  MoveL 7986 to (-27.4, 35.71, 116.27) mm, rotated rx 180 ry 0 rz 180 deg; joints [-139.207, -47.82, -97.335, 46.438, 64.37, -24.457]
  Call Extruder(71.60484)
  MoveL 7987 to (-27.15, 35.66, 116.27) mm, rotated rx 180 ry 0 rz -180 deg; joints [-139.239, -47.83, -97.308, 46.411, 64.345, -24.457]
  MoveL 7988 to (-27.15, 35.66, 116.27) mm, rotated rx 180 ry 0 rz -180 deg; joints [-139.239, -47.83, -97.308, 46.411, 64.345, -24.457]
  Call Extruder(71.75270)
  MoveL 7989 to (-26.87, 35.61, 116.27) mm, rotated rx -180 ry 0 rz -180 deg; joints [-139.275, -47.842, -97.278, 46.382, 64.317, -24.457]
  MoveL 7990 to (-26.87, 35.61, 116.27) mm, rotated rx -180 ry 0 rz -180 deg; joints [-139.275, -47.842, -97.278, 46.382, 64.317, -24.457]
  Call Extruder(71.91443)
  MoveL 7991 to (-26.57, 35.56, 116.27) mm, rotated rx 180 ry 0 rz 180 deg; joints [-139.313, -47.854, -97.243, 46.351, 64.286, -24.457]
  MoveL 7992 to (-26.57, 35.56, 116.27) mm, rotated rx 180 ry 0 rz 180 deg; joints [-139.313, -47.854, -97.243, 46.351, 64.286, -24.457]
  Call Extruder(72.07544)
  MoveL 7993 to (-26.26, 35.51, 116.27) mm, rotated rx 180 ry 0 rz 180 deg; joints [-139.351, -47.867, -97.209, 46.32, 64.255, -24.458]
  MoveL 7994 to (-26.26, 35.51, 116.27) mm, rotated rx 180 ry 0 rz 180 deg; joints [-139.351, -47.867, -97.209, 46.32, 64.255, -24.458]
  Call Extruder(72.23572)
  MoveL 7995 to (-25.96, 35.46, 116.27) mm, rotated rx 180 ry 0 rz -180 deg; joints [-139.39, -47.88, -97.174, 46.289, 64.225, -24.459]
  MoveL 7996 to (-25.96, 35.46, 116.27) mm, rotated rx 180 ry 0 rz -180 deg; joints [-139.39, -47.88, -97.174, 46.289, 64.225, -24.459]
  Call Extruder(72.39527)
  MoveL 7997 to (-25.65, 35.42, 116.27) mm, rotated rx 180 ry 0 rz 180 deg; joints [-139.428, -47.892, -97.14, 46.258, 64.194, -24.46]
  MoveL 7998 to (-25.65, 35.42, 116.27) mm, rotated rx 180 ry 0 rz 180 deg; joints [-139.428, -47.892, -97.14, 46.258, 64.194, -24.46]
  Call Extruder(72.55409)
  MoveL 7999 to (-25.34, 35.37, 116.27) mm, rotated rx 180 ry 0 rz -180 deg; joints [-139.466, -47.905, -97.105, 46.227, 64.163, -24.46]
  MoveL 8000 to (-25.34, 35.37, 116.27) mm, rotated rx 180 ry 0 rz -180 deg; joints [-139.466, -47.905, -97.105, 46.227, 64.163, -24.46]
  Call Extruder(72.73276)
  MoveL 8001 to (-25, 35.32, 116.27) mm, rotated rx 180 ry 0 rz -180 deg; joints [-139.508, -47.92, -97.065, 46.193, 64.128, -24.462]
  MoveL 8002 to (-25, 35.32, 116.27) mm, rotated rx 180 ry 0 rz -180 deg; joints [-139.508, -47.92, -97.065, 46.193, 64.128, -24.462]
  Call Extruder(72.93120)
  MoveL 8003 to (-24.61, 35.28, 116.27) mm, rotated rx 180 ry 0 rz 180 deg; joints [-139.554, -47.937, -97.019, 46.156, 64.089, -24.465]
  MoveL 8004 to (-24.61, 35.28, 116.27) mm, rotated rx 180 ry 0 rz 180 deg; joints [-139.554, -47.937, -97.019, 46.156, 64.089, -24.465]
  Call Extruder(73.12878)
  MoveL 8005 to (-24.22, 35.23, 116.27) mm, rotated rx 180 ry 0 rz 180 deg; joints [-139.6, -47.954, -96.973, 46.12, 64.05, -24.467]
  MoveL 8006 to (-24.22, 35.23, 116.27) mm, rotated rx 180 ry 0 rz 180 deg; joints [-139.6, -47.954, -96.973, 46.12, 64.05, -24.467]
  Call Extruder(73.32549)
  MoveL 8007 to (-23.84, 35.18, 116.27) mm, rotated rx -180 ry 0 rz 180 deg; joints [-139.647, -47.971, -96.928, 46.083, 64.01, -24.47]
  MoveL 8008 to (-23.84, 35.18, 116.27) mm, rotated rx -180 ry 0 rz 180 deg; joints [-139.647, -47.971, -96.928, 46.083, 64.01, -24.47]
  Call Extruder(73.52132)
  MoveL 8009 to (-23.45, 35.14, 116.27) mm, rotated rx 180 ry 0 rz 180 deg; joints [-139.693, -47.988, -96.882, 46.047, 63.971, -24.473]
  MoveL 8010 to (-23.45, 35.14, 116.27) mm, rotated rx 180 ry 0 rz 180 deg; joints [-139.693, -47.988, -96.882, 46.047, 63.971, -24.473]
  Call Extruder(73.81672)
  MoveL 8011 to (-22.86, 35.09, 116.27) mm, rotated rx 180 ry 0 rz -180 deg; joints [-139.76, -48.015, -96.809, 45.995, 63.912, -24.48]
  MoveL 8012 to (-22.86, 35.09, 116.27) mm, rotated rx 180 ry 0 rz -180 deg; joints [-139.76, -48.015, -96.809, 45.995, 63.912, -24.48]
  Call Extruder(74.11078)
  MoveL 8013 to (-22.27, 35.04, 116.27) mm, rotated rx -180 ry 0 rz -180 deg; joints [-139.826, -48.042, -96.736, 45.943, 63.852, -24.486]
  MoveL 8014 to (-22.27, 35.04, 116.27) mm, rotated rx -180 ry 0 rz -180 deg; joints [-139.826, -48.042, -96.736, 45.943, 63.852, -24.486]
  Call Extruder(74.40351)
  MoveL 8015 to (-21.68, 35, 116.27) mm, rotated rx 180 ry 0 rz 180 deg; joints [-139.893, -48.069, -96.664, 45.892, 63.793, -24.493]
  MoveL 8016 to (-21.68, 35, 116.27) mm, rotated rx 180 ry 0 rz 180 deg; joints [-139.893, -48.069, -96.664, 45.892, 63.793, -24.493]
  Call Extruder(74.97696)
  MoveL 8017 to (-20.52, 34.95, 116.27) mm, rotated rx 180 ry 0 rz -180 deg; joints [-140.019, -48.124, -96.515, 45.797, 63.675, -24.512]
  MoveL 8018 to (-20.52, 34.95, 116.27) mm, rotated rx 180 ry 0 rz -180 deg; joints [-140.019, -48.124, -96.515, 45.797, 63.675, -24.512]
  Call Extruder(75.69093)
  MoveL 8019 to (-19.06, 34.91, 116.27) mm, rotated rx 180 ry 0 rz 180 deg; joints [-140.173, -48.194, -96.326, 45.683, 63.529, -24.537]
  Call Extruder(192.53767)
  MoveL 8020 to (219.06, 34.91, 116.27) mm, rotated rx 180 ry 0 rz 180 deg; joints [-155.896, -66.609, -53.991, 41.312, 38.216, -34.626]
  Call Extruder(192.96623)
  MoveL 8021 to (219.94, 34.93, 116.27) mm, rotated rx 180 ry 0 rz -180 deg; joints [-155.931, -66.71, -53.779, 41.359, 38.112, -34.709]
  MoveL 8022 to (219.94, 34.93, 116.27) mm, rotated rx 180 ry 0 rz -180 deg; joints [-155.931, -66.71, -53.779, 41.359, 38.112, -34.709]
  Call Extruder(193.53967)
  MoveL 8023 to (221.1, 34.97, 116.27) mm, rotated rx 180 ry 0 rz 180 deg; joints [-155.975, -66.846, -53.494, 41.427, 37.975, -34.824]
  MoveL 8024 to (221.1, 34.97, 116.27) mm, rotated rx 180 ry 0 rz 180 deg; joints [-155.975, -66.846, -53.494, 41.427, 37.975, -34.824]
  Call Extruder(193.97399)
  MoveL 8025 to (221.97, 35.02, 116.27) mm, rotated rx 180 ry 0 rz 180 deg; joints [-156.007, -66.949, -53.276, 41.482, 37.871, -34.913]
  MoveL 8026 to (221.97, 35.02, 116.27) mm, rotated rx 180 ry 0 rz 180 deg; joints [-156.007, -66.949, -53.276, 41.482, 37.871, -34.913]
  Call Extruder(194.26805)
  MoveL 8027 to (222.56, 35.07, 116.27) mm, rotated rx -180 ry 0 rz -180 deg; joints [-156.027, -67.019, -53.128, 41.521, 37.802, -34.976]
  MoveL 8028 to (222.56, 35.07, 116.27) mm, rotated rx -180 ry 0 rz -180 deg; joints [-156.027, -67.019, -53.128, 41.521, 37.802, -34.976]
  Call Extruder(194.56344)
  MoveL 8029 to (223.15, 35.11, 116.27) mm, rotated rx 180 ry 0 rz 180 deg; joints [-156.047, -67.09, -52.98, 41.561, 37.732, -35.039]
  MoveL 8030 to (223.15, 35.11, 116.27) mm, rotated rx 180 ry 0 rz 180 deg; joints [-156.047, -67.09, -52.98, 41.561, 37.732, -35.039]
  Call Extruder(194.80967)
  MoveL 8031 to (223.64, 35.16, 116.27) mm, rotated rx 180 ry 0 rz 180 deg; joints [-156.062, -67.149, -52.855, 41.596, 37.674, -35.093]
  MoveL 8032 to (223.64, 35.16, 116.27) mm, rotated rx 180 ry 0 rz 180 deg; joints [-156.062, -67.149, -52.855, 41.596, 37.674, -35.093]
  Call Extruder(195.00638)
  MoveL 8033 to (224.03, 35.21, 116.27) mm, rotated rx 180 ry 0 rz 180 deg; joints [-156.074, -67.197, -52.756, 41.626, 37.628, -35.138]
  MoveL 8034 to (224.03, 35.21, 116.27) mm, rotated rx 180 ry 0 rz 180 deg; joints [-156.074, -67.197, -52.756, 41.626, 37.628, -35.138]
  Call Extruder(195.20395)
  MoveL 8035 to (224.42, 35.25, 116.27) mm, rotated rx -180 ry 0 rz 180 deg; joints [-156.086, -67.244, -52.656, 41.655, 37.583, -35.182]
  MoveL 8036 to (224.42, 35.25, 116.27) mm, rotated rx -180 ry 0 rz 180 deg; joints [-156.086, -67.244, -52.656, 41.655, 37.583, -35.182]
  Call Extruder(195.40240)
  MoveL 8037 to (224.8, 35.3, 116.27) mm, rotated rx 180 ry 0 rz 180 deg; joints [-156.097, -67.292, -52.556, 41.685, 37.537, -35.227]
  MoveL 8038 to (224.8, 35.3, 116.27) mm, rotated rx 180 ry 0 rz 180 deg; joints [-156.097, -67.292, -52.556, 41.685, 37.537, -35.227]
  Call Extruder(195.60171)
  MoveL 8039 to (225.19, 35.34, 116.27) mm, rotated rx 180 ry 0 rz 180 deg; joints [-156.109, -67.34, -52.456, 41.715, 37.491, -35.272]
  MoveL 8040 to (225.19, 35.34, 116.27) mm, rotated rx 180 ry 0 rz 180 deg; joints [-156.109, -67.34, -52.456, 41.715, 37.491, -35.272]
  Call Extruder(195.76053)
  MoveL 8041 to (225.5, 35.39, 116.27) mm, rotated rx 180 ry 0 rz 180 deg; joints [-156.117, -67.378, -52.375, 41.74, 37.455, -35.309]
  MoveL 8042 to (225.5, 35.39, 116.27) mm, rotated rx 180 ry 0 rz 180 deg; joints [-156.117, -67.378, -52.375, 41.74, 37.455, -35.309]
  Call Extruder(195.92007)
  MoveL 8043 to (225.8, 35.44, 116.27) mm, rotated rx 180 ry 0 rz 180 deg; joints [-156.125, -67.416, -52.295, 41.766, 37.419, -35.347]
  MoveL 8044 to (225.8, 35.44, 116.27) mm, rotated rx 180 ry 0 rz 180 deg; joints [-156.125, -67.416, -52.295, 41.766, 37.419, -35.347]
  Call Extruder(196.08035)
  MoveL 8045 to (226.11, 35.49, 116.27) mm, rotated rx 180 ry 0 rz 180 deg; joints [-156.133, -67.455, -52.214, 41.792, 37.383, -35.385]
  MoveL 8046 to (226.11, 35.49, 116.27) mm, rotated rx 180 ry 0 rz 180 deg; joints [-156.133, -67.455, -52.214, 41.792, 37.383, -35.385]
  Call Extruder(196.24135)
  MoveL 8047 to (226.41, 35.54, 116.27) mm, rotated rx -180 ry 0 rz -180 deg; joints [-156.141, -67.493, -52.133, 41.819, 37.347, -35.423]
  MoveL 8048 to (226.41, 35.54, 116.27) mm, rotated rx -180 ry 0 rz -180 deg; joints [-156.141, -67.493, -52.133, 41.819, 37.347, -35.423]
  Call Extruder(196.40308)
  MoveL 8049 to (226.72, 35.59, 116.27) mm, rotated rx -180 ry 0 rz -180 deg; joints [-156.149, -67.532, -52.053, 41.845, 37.311, -35.46]
  MoveL 8050 to (226.72, 35.59, 116.27) mm, rotated rx -180 ry 0 rz -180 deg; joints [-156.149, -67.532, -52.053, 41.845, 37.311, -35.46]
  Call Extruder(196.56554)
  MoveL 8051 to (227.03, 35.63, 116.27) mm, rotated rx -180 ry 0 rz 180 deg; joints [-156.157, -67.57, -51.972, 41.871, 37.275, -35.499]
  MoveL 8052 to (227.03, 35.63, 116.27) mm, rotated rx -180 ry 0 rz 180 deg; joints [-156.157, -67.57, -51.972, 41.871, 37.275, -35.499]
  Call Extruder(196.69947)
  MoveL 8053 to (227.28, 35.68, 116.27) mm, rotated rx 180 ry 0 rz 180 deg; joints [-156.162, -67.603, -51.905, 41.894, 37.245, -35.531]
  MoveL 8054 to (227.28, 35.68, 116.27) mm, rotated rx 180 ry 0 rz 180 deg; joints [-156.162, -67.603, -51.905, 41.894, 37.245, -35.531]
  Call Extruder(196.83401)
  MoveL 8055 to (227.52, 35.73, 116.27) mm, rotated rx -180 ry 0 rz -180 deg; joints [-156.168, -67.635, -51.837, 41.918, 37.216, -35.564]
  MoveL 8056 to (227.52, 35.73, 116.27) mm, rotated rx -180 ry 0 rz -180 deg; joints [-156.168, -67.635, -51.837, 41.918, 37.216, -35.564]
  Call Extruder(196.96915)
  MoveL 8057 to (227.77, 35.78, 116.27) mm, rotated rx 180 ry 0 rz -180 deg; joints [-156.173, -67.667, -51.77, 41.941, 37.186, -35.597]
  MoveL 8058 to (227.77, 35.78, 116.27) mm, rotated rx 180 ry 0 rz -180 deg; joints [-156.173, -67.667, -51.77, 41.941, 37.186, -35.597]
  Call Extruder(197.10491)
  MoveL 8059 to (228.02, 35.83, 116.27) mm, rotated rx 180 ry 0 rz 180 deg; joints [-156.179, -67.699, -51.703, 41.965, 37.157, -35.63]
  MoveL 8060 to (228.02, 35.83, 116.27) mm, rotated rx 180 ry 0 rz 180 deg; joints [-156.179, -67.699, -51.703, 41.965, 37.157, -35.63]
  Call Extruder(197.24128)
  MoveL 8061 to (228.27, 35.88, 116.27) mm, rotated rx 180 ry 0 rz 180 deg; joints [-156.185, -67.731, -51.636, 41.988, 37.128, -35.663]
  MoveL 8062 to (228.27, 35.88, 116.27) mm, rotated rx 180 ry 0 rz 180 deg; joints [-156.185, -67.731, -51.636, 41.988, 37.128, -35.663]
  Call Extruder(197.37826)
  MoveL 8063 to (228.52, 35.93, 116.27) mm, rotated rx -180 ry 0 rz 180 deg; joints [-156.19, -67.763, -51.568, 42.012, 37.098, -35.696]
  MoveL 8064 to (228.52, 35.93, 116.27) mm, rotated rx -180 ry 0 rz 180 deg; joints [-156.19, -67.763, -51.568, 42.012, 37.098, -35.696]
  Call Extruder(197.51585)
  MoveL 8065 to (228.77, 35.98, 116.27) mm, rotated rx 180 ry 0 rz 180 deg; joints [-156.196, -67.795, -51.501, 42.036, 37.069, -35.729]
  MoveL 8066 to (228.77, 35.98, 116.27) mm, rotated rx 180 ry 0 rz 180 deg; joints [-156.196, -67.795, -51.501, 42.036, 37.069, -35.729]
  Call Extruder(197.62957)
  MoveL 8067 to (228.97, 36.03, 116.27) mm, rotated rx 180 ry 0 rz 180 deg; joints [-156.2, -67.822, -51.445, 42.056, 37.045, -35.757]
  MoveL 8068 to (228.97, 36.03, 116.27) mm, rotated rx 180 ry 0 rz 180 deg; joints [-156.2, -67.822, -51.445, 42.056, 37.045, -35.757]
  Call Extruder(197.74374)
  MoveL 8069 to (229.18, 36.07, 116.27) mm, rotated rx -180 ry 0 rz 180 deg; joints [-156.204, -67.849, -51.389, 42.076, 37.021, -35.785]
  MoveL 8070 to (229.18, 36.07, 116.27) mm, rotated rx -180 ry 0 rz 180 deg; joints [-156.204, -67.849, -51.389, 42.076, 37.021, -35.785]
  Call Extruder(197.85836)
  MoveL 8071 to (229.38, 36.12, 116.27) mm, rotated rx -180 ry 0 rz 180 deg; joints [-156.208, -67.875, -51.333, 42.097, 36.997, -35.813]
  MoveL 8072 to (229.38, 36.12, 116.27) mm, rotated rx -180 ry 0 rz 180 deg; joints [-156.208, -67.875, -51.333, 42.097, 36.997, -35.813]
  Call Extruder(197.97344)
  MoveL 8073 to (229.59, 36.16, 116.27) mm, rotated rx 180 ry 0 rz 180 deg; joints [-156.212, -67.902, -51.277, 42.117, 36.973, -35.841]
  MoveL 8074 to (229.59, 36.16, 116.27) mm, rotated rx 180 ry 0 rz 180 deg; joints [-156.212, -67.902, -51.277, 42.117, 36.973, -35.841]
  Call Extruder(198.09430)
  MoveL 8075 to (229.8, 36.21, 116.27) mm, rotated rx -180 ry 0 rz 180 deg; joints [-156.216, -67.93, -51.218, 42.14, 36.948, -35.872]
  MoveL 8076 to (229.8, 36.21, 116.27) mm, rotated rx -180 ry 0 rz 180 deg; joints [-156.216, -67.93, -51.218, 42.14, 36.948, -35.872]
  Call Extruder(198.22115)
  MoveL 8077 to (230.02, 36.28, 116.27) mm, rotated rx -180 ry 0 rz -180 deg; joints [-156.219, -67.96, -51.156, 42.165, 36.922, -35.905]
  MoveL 8078 to (230.02, 36.28, 116.27) mm, rotated rx -180 ry 0 rz -180 deg; joints [-156.219, -67.96, -51.156, 42.165, 36.922, -35.905]
  Call Extruder(198.33995)
  MoveL 8079 to (230.22, 36.34, 116.27) mm, rotated rx -180 ry 0 rz -180 deg; joints [-156.222, -67.988, -51.098, 42.188, 36.898, -35.936]
  MoveL 8080 to (230.22, 36.34, 116.27) mm, rotated rx -180 ry 0 rz -180 deg; joints [-156.222, -67.988, -51.098, 42.188, 36.898, -35.936]
  Call Extruder(198.45066)
  MoveL 8081 to (230.41, 36.4, 116.27) mm, rotated rx -180 ry 0 rz -180 deg; joints [-156.224, -68.014, -51.044, 42.21, 36.876, -35.965]
  MoveL 8082 to (230.41, 36.4, 116.27) mm, rotated rx -180 ry 0 rz -180 deg; joints [-156.224, -68.014, -51.044, 42.21, 36.876, -35.965]
  Call Extruder(198.56179)
  MoveL 8083 to (230.6, 36.46, 116.27) mm, rotated rx 180 ry 0 rz -180 deg; joints [-156.226, -68.039, -50.99, 42.232, 36.854, -35.994]
  MoveL 8084 to (230.6, 36.46, 116.27) mm, rotated rx 180 ry 0 rz -180 deg; joints [-156.226, -68.039, -50.99, 42.232, 36.854, -35.994]
  Call Extruder(198.67341)
  MoveL 8085 to (230.79, 36.52, 116.27) mm, rotated rx 180 ry 0 rz 180 deg; joints [-156.228, -68.065, -50.936, 42.255, 36.831, -36.023]
  MoveL 8086 to (230.79, 36.52, 116.27) mm, rotated rx 180 ry 0 rz 180 deg; joints [-156.228, -68.065, -50.936, 42.255, 36.831, -36.023]
  Call Extruder(198.78553)
  MoveL 8087 to (230.98, 36.58, 116.27) mm, rotated rx 180 ry 0 rz 180 deg; joints [-156.23, -68.091, -50.882, 42.278, 36.809, -36.053]
  MoveL 8088 to (230.98, 36.58, 116.27) mm, rotated rx 180 ry 0 rz 180 deg; joints [-156.23, -68.091, -50.882, 42.278, 36.809, -36.053]
  Call Extruder(198.89810)
  MoveL 8089 to (231.17, 36.64, 116.27) mm, rotated rx -180 ry 0 rz 180 deg; joints [-156.232, -68.117, -50.828, 42.3, 36.787, -36.082]
  MoveL 8090 to (231.17, 36.64, 116.27) mm, rotated rx -180 ry 0 rz 180 deg; joints [-156.232, -68.117, -50.828, 42.3, 36.787, -36.082]
  Call Extruder(199.01111)
  MoveL 8091 to (231.35, 36.7, 116.27) mm, rotated rx -180 ry 0 rz 180 deg; joints [-156.234, -68.143, -50.774, 42.323, 36.765, -36.112]
  MoveL 8092 to (231.35, 36.7, 116.27) mm, rotated rx -180 ry 0 rz 180 deg; joints [-156.234, -68.143, -50.774, 42.323, 36.765, -36.112]
  Call Extruder(199.12456)
  MoveL 8093 to (231.54, 36.76, 116.27) mm, rotated rx 180 ry 0 rz -180 deg; joints [-156.236, -68.169, -50.719, 42.346, 36.743, -36.142]
  MoveL 8094 to (231.54, 36.76, 116.27) mm, rotated rx 180 ry 0 rz -180 deg; joints [-156.236, -68.169, -50.719, 42.346, 36.743, -36.142]
  Call Extruder(199.27220)
  MoveL 8095 to (231.78, 36.85, 116.27) mm, rotated rx -180 ry 0 rz 180 deg; joints [-156.237, -68.203, -50.649, 42.378, 36.715, -36.182]
  MoveL 8096 to (231.78, 36.85, 116.27) mm, rotated rx -180 ry 0 rz 180 deg; joints [-156.237, -68.203, -50.649, 42.378, 36.715, -36.182]
  Call Extruder(199.45454)
  MoveL 8097 to (232.07, 36.97, 116.27) mm, rotated rx -180 ry 0 rz 180 deg; joints [-156.238, -68.245, -50.562, 42.418, 36.681, -36.232]
  MoveL 8098 to (232.07, 36.97, 116.27) mm, rotated rx -180 ry 0 rz 180 deg; joints [-156.238, -68.245, -50.562, 42.418, 36.681, -36.232]
  Call Extruder(199.63764)
  MoveL 8099 to (232.37, 37.09, 116.27) mm, rotated rx -180 ry 0 rz 180 deg; joints [-156.239, -68.286, -50.474, 42.458, 36.647, -36.283]
  MoveL 8100 to (232.37, 37.09, 116.27) mm, rotated rx -180 ry 0 rz 180 deg; joints [-156.239, -68.286, -50.474, 42.458, 36.647, -36.283]
  Call Extruder(199.79534)
  MoveL 8101 to (232.62, 37.2, 116.27) mm, rotated rx 180 ry 0 rz 180 deg; joints [-156.239, -68.322, -50.399, 42.493, 36.618, -36.327]
  MoveL 8102 to (232.62, 37.2, 116.27) mm, rotated rx 180 ry 0 rz 180 deg; joints [-156.239, -68.322, -50.399, 42.493, 36.618, -36.327]
  Call Extruder(199.95364)
  MoveL 8103 to (232.86, 37.31, 116.27) mm, rotated rx 180 ry 0 rz 180 deg; joints [-156.239, -68.358, -50.324, 42.528, 36.589, -36.371]
  MoveL 8104 to (232.86, 37.31, 116.27) mm, rotated rx 180 ry 0 rz 180 deg; joints [-156.239, -68.358, -50.324, 42.528, 36.589, -36.371]
  Call Extruder(200.13566)
  MoveL 8105 to (233.14, 37.45, 116.27) mm, rotated rx 180 ry 0 rz 180 deg; joints [-156.237, -68.399, -50.238, 42.572, 36.557, -36.424]
  MoveL 8106 to (233.14, 37.45, 116.27) mm, rotated rx 180 ry 0 rz 180 deg; joints [-156.237, -68.399, -50.238, 42.572, 36.557, -36.424]
  Call Extruder(200.34222)
  MoveL 8107 to (233.45, 37.63, 116.27) mm, rotated rx -180 ry 0 rz -180 deg; joints [-156.234, -68.446, -50.142, 42.623, 36.522, -36.485]
  MoveL 8108 to (233.45, 37.63, 116.27) mm, rotated rx -180 ry 0 rz -180 deg; joints [-156.234, -68.446, -50.142, 42.623, 36.522, -36.485]
  Call Extruder(200.54955)
  MoveL 8109 to (233.75, 37.8, 116.27) mm, rotated rx 180 ry 0 rz -180 deg; joints [-156.23, -68.492, -50.045, 42.674, 36.488, -36.546]
  MoveL 8110 to (233.75, 37.8, 116.27) mm, rotated rx 180 ry 0 rz -180 deg; joints [-156.23, -68.492, -50.045, 42.674, 36.488, -36.546]
  Call Extruder(200.75767)
  MoveL 8111 to (234.05, 37.98, 116.27) mm, rotated rx 180 ry 0 rz -180 deg; joints [-156.226, -68.539, -49.947, 42.725, 36.453, -36.608]
  MoveL 8112 to (234.05, 37.98, 116.27) mm, rotated rx 180 ry 0 rz -180 deg; joints [-156.226, -68.539, -49.947, 42.725, 36.453, -36.608]
  Call Extruder(200.87539)
  MoveL 8113 to (234.22, 38.08, 116.27) mm, rotated rx -180 ry 0 rz -180 deg; joints [-156.224, -68.565, -49.893, 42.754, 36.433, -36.643]
  MoveL 8114 to (234.22, 38.08, 116.27) mm, rotated rx -180 ry 0 rz -180 deg; joints [-156.224, -68.565, -49.893, 42.754, 36.433, -36.643]
  Call Extruder(201.20821)
  MoveL 8115 to (234.68, 38.41, 116.27) mm, rotated rx 180 ry 0 rz -180 deg; joints [-156.212, -68.638, -49.74, 42.843, 36.382, -36.747]
  MoveL 8116 to (234.68, 38.41, 116.27) mm, rotated rx 180 ry 0 rz -180 deg; joints [-156.212, -68.638, -49.74, 42.843, 36.382, -36.747]
  Call Extruder(201.54222)
  MoveL 8117 to (235.13, 38.73, 116.27) mm, rotated rx 180 ry 0 rz -180 deg; joints [-156.201, -68.711, -49.588, 42.933, 36.331, -36.85]
  MoveL 8118 to (235.13, 38.73, 116.27) mm, rotated rx 180 ry 0 rz -180 deg; joints [-156.201, -68.711, -49.588, 42.933, 36.331, -36.85]
  Call Extruder(201.70980)
  MoveL 8119 to (235.35, 38.9, 116.27) mm, rotated rx 180 ry 0 rz -180 deg; joints [-156.195, -68.748, -49.511, 42.977, 36.305, -36.903]
  Call Extruder(202.53913)
  MoveL 8120 to (236.39, 39.81, 116.27) mm, rotated rx 180 ry 0 rz 180 deg; joints [-156.154, -68.926, -49.141, 43.212, 36.189, -37.17]
  Call Extruder(203.17020)
  MoveL 8121 to (237.09, 40.59, 116.27) mm, rotated rx 180 ry 0 rz 180 deg; joints [-156.111, -69.056, -48.871, 43.402, 36.113, -37.379]
  MoveL 8122 to (237.09, 40.59, 116.27) mm, rotated rx 180 ry 0 rz 180 deg; joints [-156.111, -69.056, -48.871, 43.402, 36.113, -37.379]
  Call Extruder(203.36780)
  MoveL 8123 to (237.3, 40.85, 116.27) mm, rotated rx 180 ry 0 rz 180 deg; joints [-156.097, -69.096, -48.787, 43.462, 36.09, -37.446]
  Call Extruder(203.70181)
  MoveL 8124 to (237.63, 41.3, 116.27) mm, rotated rx -180 ry 0 rz -180 deg; joints [-156.069, -69.162, -48.65, 43.566, 36.056, -37.559]
  MoveL 8125 to (237.63, 41.3, 116.27) mm, rotated rx -180 ry 0 rz -180 deg; joints [-156.069, -69.162, -48.65, 43.566, 36.056, -37.559]
  Call Extruder(204.03463)
  MoveL 8126 to (237.96, 41.75, 116.27) mm, rotated rx 180 ry 0 rz 180 deg; joints [-156.042, -69.228, -48.513, 43.671, 36.021, -37.672]
  MoveL 8127 to (237.96, 41.75, 116.27) mm, rotated rx 180 ry 0 rz 180 deg; joints [-156.042, -69.228, -48.513, 43.671, 36.021, -37.672]
  Call Extruder(204.21387)
  MoveL 8128 to (238.13, 41.99, 116.27) mm, rotated rx -180 ry 0 rz 180 deg; joints [-156.027, -69.264, -48.439, 43.727, 36.002, -37.734]
  MoveL 8129 to (238.13, 41.99, 116.27) mm, rotated rx -180 ry 0 rz 180 deg; joints [-156.027, -69.264, -48.439, 43.727, 36.002, -37.734]
  Call Extruder(204.42198)
  MoveL 8130 to (238.31, 42.3, 116.27) mm, rotated rx -180 ry 0 rz 180 deg; joints [-156.006, -69.303, -48.358, 43.795, 35.984, -37.805]
  MoveL 8131 to (238.31, 42.3, 116.27) mm, rotated rx -180 ry 0 rz 180 deg; joints [-156.006, -69.303, -48.358, 43.795, 35.984, -37.805]
  Call Extruder(204.62931)
  MoveL 8132 to (238.49, 42.6, 116.27) mm, rotated rx 180 ry 0 rz 180 deg; joints [-155.986, -69.342, -48.277, 43.862, 35.966, -37.877]
  MoveL 8133 to (238.49, 42.6, 116.27) mm, rotated rx 180 ry 0 rz 180 deg; joints [-155.986, -69.342, -48.277, 43.862, 35.966, -37.877]
  Call Extruder(204.83587)
  MoveL 8134 to (238.66, 42.91, 116.27) mm, rotated rx 180 ry 0 rz -180 deg; joints [-155.966, -69.381, -48.196, 43.929, 35.948, -37.949]
  MoveL 8135 to (238.66, 42.91, 116.27) mm, rotated rx 180 ry 0 rz -180 deg; joints [-155.966, -69.381, -48.196, 43.929, 35.948, -37.949]
  Call Extruder(205.04165)
  MoveL 8136 to (238.84, 43.21, 116.27) mm, rotated rx 180 ry 0 rz -180 deg; joints [-155.946, -69.42, -48.114, 43.997, 35.931, -38.02]
  MoveL 8137 to (238.84, 43.21, 116.27) mm, rotated rx 180 ry 0 rz -180 deg; joints [-155.946, -69.42, -48.114, 43.997, 35.931, -38.02]
  Call Extruder(205.19996)
  MoveL 8138 to (238.94, 43.46, 116.27) mm, rotated rx -180 ry 0 rz -180 deg; joints [-155.927, -69.447, -48.057, 44.049, 35.92, -38.075]
  MoveL 8139 to (238.94, 43.46, 116.27) mm, rotated rx -180 ry 0 rz -180 deg; joints [-155.927, -69.447, -48.057, 44.049, 35.92, -38.075]
  Call Extruder(205.35767)
  MoveL 8140 to (239.05, 43.71, 116.27) mm, rotated rx 180 ry 0 rz 180 deg; joints [-155.909, -69.475, -48, 44.102, 35.91, -38.13]
  MoveL 8141 to (239.05, 43.71, 116.27) mm, rotated rx 180 ry 0 rz 180 deg; joints [-155.909, -69.475, -48, 44.102, 35.91, -38.13]
  Call Extruder(205.52776)
  MoveL 8142 to (239.17, 43.98, 116.27) mm, rotated rx 180 ry 0 rz 180 deg; joints [-155.89, -69.505, -47.939, 44.159, 35.9, -38.189]
  MoveL 8143 to (239.17, 43.98, 116.27) mm, rotated rx 180 ry 0 rz 180 deg; joints [-155.89, -69.505, -47.939, 44.159, 35.9, -38.189]
  Call Extruder(205.71010)
  MoveL 8144 to (239.29, 44.27, 116.27) mm, rotated rx -180 ry 0 rz -180 deg; joints [-155.869, -69.536, -47.873, 44.22, 35.888, -38.252]
  MoveL 8145 to (239.29, 44.27, 116.27) mm, rotated rx -180 ry 0 rz -180 deg; joints [-155.869, -69.536, -47.873, 44.22, 35.888, -38.252]
  Call Extruder(205.89168)
  MoveL 8146 to (239.41, 44.56, 116.27) mm, rotated rx 180 ry 0 rz 180 deg; joints [-155.847, -69.568, -47.807, 44.282, 35.877, -38.316]
  MoveL 8147 to (239.41, 44.56, 116.27) mm, rotated rx 180 ry 0 rz 180 deg; joints [-155.847, -69.568, -47.807, 44.282, 35.877, -38.316]
  Call Extruder(206.00513)
  MoveL 8148 to (239.47, 44.75, 116.27) mm, rotated rx 180 ry 0 rz -180 deg; joints [-155.833, -69.587, -47.769, 44.32, 35.872, -38.355]
  MoveL 8149 to (239.47, 44.75, 116.27) mm, rotated rx 180 ry 0 rz -180 deg; joints [-155.833, -69.587, -47.769, 44.32, 35.872, -38.355]
  Call Extruder(206.11815)
  MoveL 8150 to (239.53, 44.94, 116.27) mm, rotated rx -180 ry 0 rz 180 deg; joints [-155.819, -69.605, -47.73, 44.358, 35.866, -38.395]
  MoveL 8151 to (239.53, 44.94, 116.27) mm, rotated rx -180 ry 0 rz 180 deg; joints [-155.819, -69.605, -47.73, 44.358, 35.866, -38.395]
  Call Extruder(206.23072)
  MoveL 8152 to (239.59, 45.13, 116.27) mm, rotated rx 180 ry 0 rz 180 deg; joints [-155.804, -69.624, -47.692, 44.397, 35.861, -38.434]
  MoveL 8153 to (239.59, 45.13, 116.27) mm, rotated rx 180 ry 0 rz 180 deg; joints [-155.804, -69.624, -47.692, 44.397, 35.861, -38.434]
  Call Extruder(206.34284)
  MoveL 8154 to (239.65, 45.32, 116.27) mm, rotated rx -180 ry 0 rz 180 deg; joints [-155.79, -69.642, -47.654, 44.435, 35.856, -38.473]
  MoveL 8155 to (239.65, 45.32, 116.27) mm, rotated rx -180 ry 0 rz 180 deg; joints [-155.79, -69.642, -47.654, 44.435, 35.856, -38.473]
  Call Extruder(206.45452)
  MoveL 8156 to (239.71, 45.5, 116.27) mm, rotated rx -180 ry 0 rz 180 deg; joints [-155.776, -69.66, -47.615, 44.474, 35.851, -38.513]
  MoveL 8157 to (239.71, 45.5, 116.27) mm, rotated rx -180 ry 0 rz 180 deg; joints [-155.776, -69.66, -47.615, 44.474, 35.851, -38.513]
  Call Extruder(206.58559)
  MoveL 8158 to (239.78, 45.73, 116.27) mm, rotated rx 180 ry 0 rz 180 deg; joints [-155.758, -69.682, -47.571, 44.519, 35.845, -38.559]
  MoveL 8159 to (239.78, 45.73, 116.27) mm, rotated rx 180 ry 0 rz 180 deg; joints [-155.758, -69.682, -47.571, 44.519, 35.845, -38.559]
  Call Extruder(206.71610)
  MoveL 8160 to (239.85, 45.95, 116.27) mm, rotated rx -180 ry 0 rz 180 deg; joints [-155.741, -69.703, -47.527, 44.564, 35.839, -38.605]
  MoveL 8161 to (239.85, 45.95, 116.27) mm, rotated rx -180 ry 0 rz 180 deg; joints [-155.741, -69.703, -47.527, 44.564, 35.839, -38.605]
  Call Extruder(206.84604)
  MoveL 8162 to (239.92, 46.18, 116.27) mm, rotated rx -180 ry 0 rz 180 deg; joints [-155.724, -69.725, -47.482, 44.61, 35.834, -38.651]
  MoveL 8163 to (239.92, 46.18, 116.27) mm, rotated rx -180 ry 0 rz 180 deg; joints [-155.724, -69.725, -47.482, 44.61, 35.834, -38.651]
  Call Extruder(206.97542)
  MoveL 8164 to (239.98, 46.4, 116.27) mm, rotated rx -180 ry 0 rz 180 deg; joints [-155.707, -69.746, -47.438, 44.655, 35.828, -38.697]
  MoveL 8165 to (239.98, 46.4, 116.27) mm, rotated rx -180 ry 0 rz 180 deg; joints [-155.707, -69.746, -47.438, 44.655, 35.828, -38.697]
  Call Extruder(207.09738)
  MoveL 8166 to (240.04, 46.61, 116.27) mm, rotated rx 180 ry 0 rz -180 deg; joints [-155.69, -69.766, -47.397, 44.698, 35.824, -38.74]
  MoveL 8167 to (240.04, 46.61, 116.27) mm, rotated rx 180 ry 0 rz -180 deg; joints [-155.69, -69.766, -47.397, 44.698, 35.824, -38.74]
  Call Extruder(207.21220)
  MoveL 8168 to (240.08, 46.82, 116.27) mm, rotated rx 180 ry 0 rz 180 deg; joints [-155.674, -69.783, -47.362, 44.738, 35.821, -38.78]
  MoveL 8169 to (240.08, 46.82, 116.27) mm, rotated rx 180 ry 0 rz 180 deg; joints [-155.674, -69.783, -47.362, 44.738, 35.821, -38.78]
  Call Extruder(207.32658)
  MoveL 8170 to (240.13, 47.02, 116.27) mm, rotated rx 180 ry 0 rz 180 deg; joints [-155.657, -69.8, -47.325, 44.778, 35.818, -38.821]
  MoveL 8171 to (240.13, 47.02, 116.27) mm, rotated rx 180 ry 0 rz 180 deg; joints [-155.657, -69.8, -47.325, 44.778, 35.818, -38.821]
  Call Extruder(207.44050)
  MoveL 8172 to (240.17, 47.23, 116.27) mm, rotated rx 180 ry 0 rz -180 deg; joints [-155.641, -69.818, -47.289, 44.818, 35.815, -38.861]
  MoveL 8173 to (240.17, 47.23, 116.27) mm, rotated rx 180 ry 0 rz -180 deg; joints [-155.641, -69.818, -47.289, 44.818, 35.815, -38.861]
  Call Extruder(207.55397)
  MoveL 8174 to (240.22, 47.43, 116.27) mm, rotated rx 180 ry 0 rz 180 deg; joints [-155.624, -69.835, -47.253, 44.858, 35.812, -38.901]
  MoveL 8175 to (240.22, 47.43, 116.27) mm, rotated rx 180 ry 0 rz 180 deg; joints [-155.624, -69.835, -47.253, 44.858, 35.812, -38.901]
  Call Extruder(207.69125)
  MoveL 8176 to (240.27, 47.68, 116.27) mm, rotated rx -180 ry 0 rz 180 deg; joints [-155.604, -69.856, -47.21, 44.906, 35.809, -38.95]
  MoveL 8177 to (240.27, 47.68, 116.27) mm, rotated rx -180 ry 0 rz 180 deg; joints [-155.604, -69.856, -47.21, 44.906, 35.809, -38.95]
  Call Extruder(207.82792)
  MoveL 8178 to (240.32, 47.93, 116.27) mm, rotated rx -180 ry 0 rz 180 deg; joints [-155.584, -69.877, -47.167, 44.955, 35.806, -38.998]
  MoveL 8179 to (240.32, 47.93, 116.27) mm, rotated rx -180 ry 0 rz 180 deg; joints [-155.584, -69.877, -47.167, 44.955, 35.806, -38.998]
  Call Extruder(207.96399)
  MoveL 8180 to (240.37, 48.18, 116.27) mm, rotated rx 180 ry 0 rz 180 deg; joints [-155.564, -69.897, -47.124, 45.003, 35.802, -39.047]
  MoveL 8181 to (240.37, 48.18, 116.27) mm, rotated rx 180 ry 0 rz 180 deg; joints [-155.564, -69.897, -47.124, 45.003, 35.802, -39.047]
  Call Extruder(208.09944)
  MoveL 8182 to (240.42, 48.43, 116.27) mm, rotated rx 180 ry 0 rz 180 deg; joints [-155.544, -69.918, -47.081, 45.052, 35.799, -39.095]
  MoveL 8183 to (240.42, 48.43, 116.27) mm, rotated rx 180 ry 0 rz 180 deg; joints [-155.544, -69.918, -47.081, 45.052, 35.799, -39.095]
  Call Extruder(208.23428)
  MoveL 8184 to (240.47, 48.68, 116.27) mm, rotated rx 180 ry 0 rz 180 deg; joints [-155.524, -69.939, -47.038, 45.1, 35.796, -39.144]
  MoveL 8185 to (240.47, 48.68, 116.27) mm, rotated rx 180 ry 0 rz 180 deg; joints [-155.524, -69.939, -47.038, 45.1, 35.796, -39.144]
  Call Extruder(208.36851)
  MoveL 8186 to (240.52, 48.92, 116.27) mm, rotated rx -180 ry 0 rz 180 deg; joints [-155.504, -69.96, -46.995, 45.149, 35.793, -39.192]
  MoveL 8187 to (240.52, 48.92, 116.27) mm, rotated rx -180 ry 0 rz 180 deg; joints [-155.504, -69.96, -46.995, 45.149, 35.793, -39.192]
  Call Extruder(208.50213)
  MoveL 8188 to (240.56, 49.17, 116.27) mm, rotated rx 180 ry 0 rz -180 deg; joints [-155.484, -69.981, -46.952, 45.197, 35.79, -39.241]
  MoveL 8189 to (240.56, 49.17, 116.27) mm, rotated rx 180 ry 0 rz -180 deg; joints [-155.484, -69.981, -46.952, 45.197, 35.79, -39.241]
  Call Extruder(208.66424)
  MoveL 8190 to (240.61, 49.48, 116.27) mm, rotated rx 180 ry 0 rz 180 deg; joints [-155.459, -70.005, -46.902, 45.256, 35.788, -39.299]
  MoveL 8191 to (240.61, 49.48, 116.27) mm, rotated rx 180 ry 0 rz 180 deg; joints [-155.459, -70.005, -46.902, 45.256, 35.788, -39.299]
  Call Extruder(208.82562)
  MoveL 8192 to (240.66, 49.79, 116.27) mm, rotated rx 180 ry 0 rz 180 deg; joints [-155.433, -70.029, -46.852, 45.315, 35.786, -39.358]
  MoveL 8193 to (240.66, 49.79, 116.27) mm, rotated rx 180 ry 0 rz 180 deg; joints [-155.433, -70.029, -46.852, 45.315, 35.786, -39.358]
  Call Extruder(208.98628)
  MoveL 8194 to (240.71, 50.09, 116.27) mm, rotated rx -180 ry 0 rz 180 deg; joints [-155.408, -70.053, -46.802, 45.374, 35.783, -39.416]
  MoveL 8195 to (240.71, 50.09, 116.27) mm, rotated rx -180 ry 0 rz 180 deg; joints [-155.408, -70.053, -46.802, 45.374, 35.783, -39.416]
  Call Extruder(209.14620)
  MoveL 8196 to (240.76, 50.4, 116.27) mm, rotated rx 180 ry 0 rz 180 deg; joints [-155.383, -70.077, -46.752, 45.432, 35.781, -39.474]
  MoveL 8197 to (240.76, 50.4, 116.27) mm, rotated rx 180 ry 0 rz 180 deg; joints [-155.383, -70.077, -46.752, 45.432, 35.781, -39.474]
  Call Extruder(209.30540)
  MoveL 8198 to (240.81, 50.7, 116.27) mm, rotated rx 180 ry 0 rz 180 deg; joints [-155.358, -70.102, -46.701, 45.491, 35.779, -39.533]
  MoveL 8199 to (240.81, 50.7, 116.27) mm, rotated rx 180 ry 0 rz 180 deg; joints [-155.358, -70.102, -46.701, 45.491, 35.779, -39.533]
  Call Extruder(209.46387)
  MoveL 8200 to (240.86, 51.01, 116.27) mm, rotated rx 180 ry 0 rz 180 deg; joints [-155.333, -70.126, -46.651, 45.55, 35.777, -39.591]
  MoveL 8201 to (240.86, 51.01, 116.27) mm, rotated rx 180 ry 0 rz 180 deg; joints [-155.333, -70.126, -46.651, 45.55, 35.777, -39.591]
  Call Extruder(209.66274)
  MoveL 8202 to (240.9, 51.4, 116.27) mm, rotated rx 180 ry 0 rz -180 deg; joints [-155.301, -70.155, -46.592, 45.623, 35.776, -39.663]
  MoveL 8203 to (240.9, 51.4, 116.27) mm, rotated rx 180 ry 0 rz -180 deg; joints [-155.301, -70.155, -46.592, 45.623, 35.776, -39.663]
  Call Extruder(209.86075)
  MoveL 8204 to (240.95, 51.78, 116.27) mm, rotated rx -180 ry 0 rz 180 deg; joints [-155.268, -70.184, -46.532, 45.696, 35.775, -39.736]
  MoveL 8205 to (240.95, 51.78, 116.27) mm, rotated rx -180 ry 0 rz 180 deg; joints [-155.268, -70.184, -46.532, 45.696, 35.775, -39.736]
  Call Extruder(210.05789)
  MoveL 8206 to (240.99, 52.17, 116.27) mm, rotated rx -180 ry 0 rz 180 deg; joints [-155.236, -70.212, -46.472, 45.769, 35.774, -39.808]
  MoveL 8207 to (240.99, 52.17, 116.27) mm, rotated rx -180 ry 0 rz 180 deg; joints [-155.236, -70.212, -46.472, 45.769, 35.774, -39.808]
  Call Extruder(210.25416)
  MoveL 8208 to (241.04, 52.56, 116.27) mm, rotated rx 180 ry 0 rz -180 deg; joints [-155.204, -70.241, -46.412, 45.842, 35.773, -39.881]
  MoveL 8209 to (241.04, 52.56, 116.27) mm, rotated rx 180 ry 0 rz -180 deg; joints [-155.204, -70.241, -46.412, 45.842, 35.773, -39.881]
  Call Extruder(210.49987)
  MoveL 8210 to (241.09, 53.05, 116.27) mm, rotated rx -180 ry 0 rz 180 deg; joints [-155.163, -70.276, -46.34, 45.934, 35.774, -39.97]
  MoveL 8211 to (241.09, 53.05, 116.27) mm, rotated rx -180 ry 0 rz 180 deg; joints [-155.163, -70.276, -46.34, 45.934, 35.774, -39.97]
  Call Extruder(210.79465)
  MoveL 8212 to (241.13, 53.64, 116.27) mm, rotated rx 180 ry 0 rz 180 deg; joints [-155.113, -70.318, -46.254, 46.043, 35.775, -40.078]
  MoveL 8213 to (241.13, 53.64, 116.27) mm, rotated rx 180 ry 0 rz 180 deg; joints [-155.113, -70.318, -46.254, 46.043, 35.775, -40.078]
  Call Extruder(211.08809)
  MoveL 8214 to (241.18, 54.23, 116.27) mm, rotated rx 180 ry 0 rz 180 deg; joints [-155.063, -70.359, -46.169, 46.153, 35.777, -40.185]
  MoveL 8215 to (241.18, 54.23, 116.27) mm, rotated rx 180 ry 0 rz 180 deg; joints [-155.063, -70.359, -46.169, 46.153, 35.777, -40.185]
  Call Extruder(211.52144)
  MoveL 8216 to (241.22, 55.1, 116.27) mm, rotated rx 180 ry 0 rz -180 deg; joints [-154.988, -70.418, -46.047, 46.314, 35.782, -40.342]
  MoveL 8217 to (241.22, 55.1, 116.27) mm, rotated rx 180 ry 0 rz -180 deg; joints [-154.988, -70.418, -46.047, 46.314, 35.782, -40.342]
  Call Extruder(212.09360)
  MoveL 8218 to (241.27, 56.26, 116.27) mm, rotated rx -180 ry 0 rz 180 deg; joints [-154.887, -70.494, -45.889, 46.526, 35.791, -40.549]
  MoveL 8219 to (241.27, 56.26, 116.27) mm, rotated rx -180 ry 0 rz 180 deg; joints [-154.887, -70.494, -45.889, 46.526, 35.791, -40.549]
  Call Extruder(212.52130)
  MoveL 8220 to (241.29, 57.14, 116.27) mm, rotated rx 180 ry 0 rz 180 deg; joints [-154.812, -70.55, -45.775, 46.684, 35.799, -40.702]
  Call Extruder(254.51494)
  MoveL 8221 to (241.29, 142.86, 116.27) mm, rotated rx 180 ry 0 rz 180 deg; joints [-147.778, -77.31, -32.008, 62.307, 37.026, -56.678]
  MoveL 8222 to (241.29, 142.86, 116.27) mm, rotated rx 180 ry 0 rz 180 deg; joints [-147.778, -77.31, -32.008, 62.307, 37.026, -56.678]
  Call Extruder(255.23038)
  MoveL 8223 to (241.25, 144.32, 116.27) mm, rotated rx 180 ry 0 rz -180 deg; joints [-147.665, -77.452, -31.723, 62.578, 37.055, -56.971]
  MoveL 8224 to (241.25, 144.32, 116.27) mm, rotated rx 180 ry 0 rz -180 deg; joints [-147.665, -77.452, -31.723, 62.578, 37.055, -56.971]
  Call Extruder(255.80512)
  MoveL 8225 to (241.2, 145.48, 116.27) mm, rotated rx 180 ry 0 rz 180 deg; joints [-147.574, -77.564, -31.498, 62.792, 37.079, -57.203]
  MoveL 8226 to (241.2, 145.48, 116.27) mm, rotated rx 180 ry 0 rz 180 deg; joints [-147.574, -77.564, -31.498, 62.792, 37.079, -57.203]
  Call Extruder(256.09856)
  MoveL 8227 to (241.16, 146.07, 116.27) mm, rotated rx 180 ry 0 rz 180 deg; joints [-147.527, -77.617, -31.391, 62.898, 37.094, -57.316]
  MoveL 8228 to (241.16, 146.07, 116.27) mm, rotated rx 180 ry 0 rz 180 deg; joints [-147.527, -77.617, -31.391, 62.898, 37.094, -57.316]
  Call Extruder(256.39333)
  MoveL 8229 to (241.11, 146.66, 116.27) mm, rotated rx -180 ry 0 rz -180 deg; joints [-147.48, -77.671, -31.283, 63.004, 37.109, -57.429]
  MoveL 8230 to (241.11, 146.66, 116.27) mm, rotated rx -180 ry 0 rz -180 deg; joints [-147.48, -77.671, -31.283, 63.004, 37.109, -57.429]
  Call Extruder(256.68944)
  MoveL 8231 to (241.06, 147.25, 116.27) mm, rotated rx -180 ry 0 rz 180 deg; joints [-147.433, -77.724, -31.175, 63.11, 37.124, -57.543]
  MoveL 8232 to (241.06, 147.25, 116.27) mm, rotated rx -180 ry 0 rz 180 deg; joints [-147.433, -77.724, -31.175, 63.11, 37.124, -57.543]
  Call Extruder(256.88571)
  MoveL 8233 to (241.02, 147.63, 116.27) mm, rotated rx 180 ry 0 rz 180 deg; joints [-147.401, -77.758, -31.109, 63.177, 37.136, -57.614]
  MoveL 8234 to (241.02, 147.63, 116.27) mm, rotated rx 180 ry 0 rz 180 deg; joints [-147.401, -77.758, -31.109, 63.177, 37.136, -57.614]
  Call Extruder(257.08285)
  MoveL 8235 to (240.97, 148.02, 116.27) mm, rotated rx 180 ry 0 rz 180 deg; joints [-147.37, -77.791, -31.042, 63.244, 37.148, -57.686]
  MoveL 8236 to (240.97, 148.02, 116.27) mm, rotated rx 180 ry 0 rz 180 deg; joints [-147.37, -77.791, -31.042, 63.244, 37.148, -57.686]
  Call Extruder(257.28085)
  MoveL 8237 to (240.92, 148.41, 116.27) mm, rotated rx 180 ry 0 rz -180 deg; joints [-147.338, -77.824, -30.976, 63.311, 37.159, -57.757]
  MoveL 8238 to (240.92, 148.41, 116.27) mm, rotated rx 180 ry 0 rz -180 deg; joints [-147.338, -77.824, -30.976, 63.311, 37.159, -57.757]
  Call Extruder(257.47973)
  MoveL 8239 to (240.88, 148.8, 116.27) mm, rotated rx -180 ry 0 rz -180 deg; joints [-147.306, -77.857, -30.909, 63.379, 37.171, -57.829]
  MoveL 8240 to (240.88, 148.8, 116.27) mm, rotated rx -180 ry 0 rz -180 deg; joints [-147.306, -77.857, -30.909, 63.379, 37.171, -57.829]
  Call Extruder(257.65881)
  MoveL 8241 to (240.83, 149.14, 116.27) mm, rotated rx 180 ry 0 rz 180 deg; joints [-147.278, -77.886, -30.851, 63.438, 37.182, -57.892]
  MoveL 8242 to (240.83, 149.14, 116.27) mm, rotated rx 180 ry 0 rz 180 deg; joints [-147.278, -77.886, -30.851, 63.438, 37.182, -57.892]
  Call Extruder(257.81801)
  MoveL 8243 to (240.78, 149.45, 116.27) mm, rotated rx -180 ry 0 rz 180 deg; joints [-147.252, -77.91, -30.802, 63.489, 37.193, -57.946]
  MoveL 8244 to (240.78, 149.45, 116.27) mm, rotated rx -180 ry 0 rz 180 deg; joints [-147.252, -77.91, -30.802, 63.489, 37.193, -57.946]
  Call Extruder(257.97794)
  MoveL 8245 to (240.74, 149.76, 116.27) mm, rotated rx 180 ry 0 rz -180 deg; joints [-147.227, -77.935, -30.753, 63.541, 37.204, -58]
  MoveL 8246 to (240.74, 149.76, 116.27) mm, rotated rx 180 ry 0 rz -180 deg; joints [-147.227, -77.935, -30.753, 63.541, 37.204, -58]
  Call Extruder(258.13859)
  MoveL 8247 to (240.69, 150.06, 116.27) mm, rotated rx -180 ry 0 rz 180 deg; joints [-147.201, -77.959, -30.704, 63.592, 37.214, -58.054]
  MoveL 8248 to (240.69, 150.06, 116.27) mm, rotated rx -180 ry 0 rz 180 deg; joints [-147.201, -77.959, -30.704, 63.592, 37.214, -58.054]
  Call Extruder(258.29997)
  MoveL 8249 to (240.64, 150.37, 116.27) mm, rotated rx 180 ry 0 rz 180 deg; joints [-147.176, -77.983, -30.655, 63.643, 37.225, -58.109]
  MoveL 8250 to (240.64, 150.37, 116.27) mm, rotated rx 180 ry 0 rz 180 deg; joints [-147.176, -77.983, -30.655, 63.643, 37.225, -58.109]
  Call Extruder(258.46208)
  MoveL 8251 to (240.59, 150.67, 116.27) mm, rotated rx -180 ry 0 rz 180 deg; joints [-147.15, -78.008, -30.606, 63.695, 37.236, -58.163]
  MoveL 8252 to (240.59, 150.67, 116.27) mm, rotated rx -180 ry 0 rz 180 deg; joints [-147.15, -78.008, -30.606, 63.695, 37.236, -58.163]
  Call Extruder(258.61028)
  MoveL 8253 to (240.54, 150.95, 116.27) mm, rotated rx -180 ry 0 rz 180 deg; joints [-147.127, -78.029, -30.563, 63.74, 37.246, -58.211]
  MoveL 8254 to (240.54, 150.95, 116.27) mm, rotated rx -180 ry 0 rz 180 deg; joints [-147.127, -78.029, -30.563, 63.74, 37.246, -58.211]
  Call Extruder(258.74452)
  MoveL 8255 to (240.49, 151.2, 116.27) mm, rotated rx 180 ry 0 rz 180 deg; joints [-147.106, -78.048, -30.526, 63.781, 37.256, -58.253]
  MoveL 8256 to (240.49, 151.2, 116.27) mm, rotated rx 180 ry 0 rz 180 deg; joints [-147.106, -78.048, -30.526, 63.781, 37.256, -58.253]
  Call Extruder(258.87936)
  MoveL 8257 to (240.44, 151.45, 116.27) mm, rotated rx -180 ry 0 rz -180 deg; joints [-147.085, -78.066, -30.489, 63.821, 37.266, -58.295]
  MoveL 8258 to (240.44, 151.45, 116.27) mm, rotated rx -180 ry 0 rz -180 deg; joints [-147.085, -78.066, -30.489, 63.821, 37.266, -58.295]
  Call Extruder(259.01481)
  MoveL 8259 to (240.39, 151.7, 116.27) mm, rotated rx -180 ry 0 rz -180 deg; joints [-147.064, -78.085, -30.452, 63.861, 37.275, -58.338]
  MoveL 8260 to (240.39, 151.7, 116.27) mm, rotated rx -180 ry 0 rz -180 deg; joints [-147.064, -78.085, -30.452, 63.861, 37.275, -58.338]
  Call Extruder(259.15087)
  MoveL 8261 to (240.34, 151.95, 116.27) mm, rotated rx -180 ry 0 rz 180 deg; joints [-147.042, -78.103, -30.415, 63.902, 37.285, -58.38]
  MoveL 8262 to (240.34, 151.95, 116.27) mm, rotated rx -180 ry 0 rz 180 deg; joints [-147.042, -78.103, -30.415, 63.902, 37.285, -58.38]
  Call Extruder(259.28754)
  MoveL 8263 to (240.29, 152.2, 116.27) mm, rotated rx 180 ry 0 rz 180 deg; joints [-147.021, -78.122, -30.377, 63.942, 37.295, -58.422]
  MoveL 8264 to (240.29, 152.2, 116.27) mm, rotated rx 180 ry 0 rz 180 deg; joints [-147.021, -78.122, -30.377, 63.942, 37.295, -58.422]
  Call Extruder(259.42483)
  MoveL 8265 to (240.24, 152.44, 116.27) mm, rotated rx -180 ry 0 rz 180 deg; joints [-147, -78.141, -30.34, 63.982, 37.305, -58.465]
  MoveL 8266 to (240.24, 152.44, 116.27) mm, rotated rx -180 ry 0 rz 180 deg; joints [-147, -78.141, -30.34, 63.982, 37.305, -58.465]
  Call Extruder(259.55049)
  MoveL 8267 to (240.2, 152.67, 116.27) mm, rotated rx -180 ry 0 rz 180 deg; joints [-146.981, -78.157, -30.307, 64.019, 37.314, -58.502]
  MoveL 8268 to (240.2, 152.67, 116.27) mm, rotated rx -180 ry 0 rz 180 deg; joints [-146.981, -78.157, -30.307, 64.019, 37.314, -58.502]
  Call Extruder(259.66441)
  MoveL 8269 to (240.15, 152.88, 116.27) mm, rotated rx -180 ry 0 rz 180 deg; joints [-146.963, -78.172, -30.278, 64.051, 37.323, -58.536]
  MoveL 8270 to (240.15, 152.88, 116.27) mm, rotated rx -180 ry 0 rz 180 deg; joints [-146.963, -78.172, -30.278, 64.051, 37.323, -58.536]
  Call Extruder(259.77879)
  MoveL 8271 to (240.11, 153.08, 116.27) mm, rotated rx 180 ry 0 rz -180 deg; joints [-146.945, -78.187, -30.248, 64.084, 37.331, -58.57]
  MoveL 8272 to (240.11, 153.08, 116.27) mm, rotated rx 180 ry 0 rz -180 deg; joints [-146.945, -78.187, -30.248, 64.084, 37.331, -58.57]
  Call Extruder(259.89362)
  MoveL 8273 to (240.06, 153.28, 116.27) mm, rotated rx 180 ry 0 rz 180 deg; joints [-146.928, -78.201, -30.219, 64.116, 37.34, -58.604]
  MoveL 8274 to (240.06, 153.28, 116.27) mm, rotated rx 180 ry 0 rz 180 deg; joints [-146.928, -78.201, -30.219, 64.116, 37.34, -58.604]
  Call Extruder(260.00890)
  MoveL 8275 to (240.02, 153.49, 116.27) mm, rotated rx 180 ry 0 rz -180 deg; joints [-146.91, -78.216, -30.189, 64.149, 37.348, -58.638]
  MoveL 8276 to (240.02, 153.49, 116.27) mm, rotated rx 180 ry 0 rz -180 deg; joints [-146.91, -78.216, -30.189, 64.149, 37.348, -58.638]
  Call Extruder(260.13828)
  MoveL 8277 to (239.95, 153.71, 116.27) mm, rotated rx -180 ry 0 rz 180 deg; joints [-146.89, -78.229, -30.163, 64.181, 37.36, -58.671]
  MoveL 8278 to (239.95, 153.71, 116.27) mm, rotated rx -180 ry 0 rz 180 deg; joints [-146.89, -78.229, -30.163, 64.181, 37.36, -58.671]
  Call Extruder(260.26822)
  MoveL 8279 to (239.88, 153.94, 116.27) mm, rotated rx 180 ry 0 rz -180 deg; joints [-146.87, -78.242, -30.137, 64.214, 37.371, -58.704]
  MoveL 8280 to (239.88, 153.94, 116.27) mm, rotated rx 180 ry 0 rz -180 deg; joints [-146.87, -78.242, -30.137, 64.214, 37.371, -58.704]
  Call Extruder(260.39873)
  MoveL 8281 to (239.82, 154.16, 116.27) mm, rotated rx 180 ry 0 rz 180 deg; joints [-146.85, -78.255, -30.111, 64.247, 37.383, -58.737]
  MoveL 8282 to (239.82, 154.16, 116.27) mm, rotated rx 180 ry 0 rz 180 deg; joints [-146.85, -78.255, -30.111, 64.247, 37.383, -58.737]
  Call Extruder(260.52980)
  MoveL 8283 to (239.75, 154.38, 116.27) mm, rotated rx 180 ry 0 rz 180 deg; joints [-146.83, -78.268, -30.085, 64.279, 37.394, -58.77]
  MoveL 8284 to (239.75, 154.38, 116.27) mm, rotated rx 180 ry 0 rz 180 deg; joints [-146.83, -78.268, -30.085, 64.279, 37.394, -58.77]
  Call Extruder(260.65144)
  MoveL 8285 to (239.68, 154.59, 116.27) mm, rotated rx 180 ry 0 rz 180 deg; joints [-146.811, -78.28, -30.061, 64.309, 37.405, -58.8]
  MoveL 8286 to (239.68, 154.59, 116.27) mm, rotated rx 180 ry 0 rz 180 deg; joints [-146.811, -78.28, -30.061, 64.309, 37.405, -58.8]
  Call Extruder(260.76357)
  MoveL 8287 to (239.62, 154.78, 116.27) mm, rotated rx 180 ry 0 rz 180 deg; joints [-146.794, -78.29, -30.041, 64.336, 37.416, -58.827]
  MoveL 8288 to (239.62, 154.78, 116.27) mm, rotated rx 180 ry 0 rz 180 deg; joints [-146.794, -78.29, -30.041, 64.336, 37.416, -58.827]
  Call Extruder(260.87613)
  MoveL 8289 to (239.56, 154.97, 116.27) mm, rotated rx 180 ry 0 rz 180 deg; joints [-146.777, -78.3, -30.02, 64.363, 37.426, -58.854]
  MoveL 8290 to (239.56, 154.97, 116.27) mm, rotated rx 180 ry 0 rz 180 deg; joints [-146.777, -78.3, -30.02, 64.363, 37.426, -58.854]
  Call Extruder(260.98915)
  MoveL 8291 to (239.5, 155.15, 116.27) mm, rotated rx 180 ry 0 rz 180 deg; joints [-146.76, -78.311, -29.999, 64.39, 37.436, -58.881]
  MoveL 8292 to (239.5, 155.15, 116.27) mm, rotated rx 180 ry 0 rz 180 deg; joints [-146.76, -78.311, -29.999, 64.39, 37.436, -58.881]
  Call Extruder(261.10260)
  MoveL 8293 to (239.44, 155.34, 116.27) mm, rotated rx 180 ry 0 rz -180 deg; joints [-146.742, -78.321, -29.978, 64.416, 37.446, -58.908]
  MoveL 8294 to (239.44, 155.34, 116.27) mm, rotated rx 180 ry 0 rz -180 deg; joints [-146.742, -78.321, -29.978, 64.416, 37.446, -58.908]
  Call Extruder(261.25025)
  MoveL 8295 to (239.35, 155.58, 116.27) mm, rotated rx 180 ry 0 rz 180 deg; joints [-146.72, -78.332, -29.956, 64.449, 37.461, -58.94]
  MoveL 8296 to (239.35, 155.58, 116.27) mm, rotated rx 180 ry 0 rz 180 deg; joints [-146.72, -78.332, -29.956, 64.449, 37.461, -58.94]
  Call Extruder(261.43258)
  MoveL 8297 to (239.22, 155.87, 116.27) mm, rotated rx 180 ry 0 rz 180 deg; joints [-146.692, -78.344, -29.932, 64.486, 37.479, -58.976]
  MoveL 8298 to (239.22, 155.87, 116.27) mm, rotated rx 180 ry 0 rz 180 deg; joints [-146.692, -78.344, -29.932, 64.486, 37.479, -58.976]
  Call Extruder(261.61568)
  MoveL 8299 to (239.1, 156.17, 116.27) mm, rotated rx -180 ry 0 rz 180 deg; joints [-146.664, -78.356, -29.908, 64.524, 37.498, -59.013]
  MoveL 8300 to (239.1, 156.17, 116.27) mm, rotated rx -180 ry 0 rz 180 deg; joints [-146.664, -78.356, -29.908, 64.524, 37.498, -59.013]
  Call Extruder(261.77338)
  MoveL 8301 to (239, 156.42, 116.27) mm, rotated rx 180 ry 0 rz -180 deg; joints [-146.64, -78.365, -29.889, 64.555, 37.514, -59.043]
  MoveL 8302 to (239, 156.42, 116.27) mm, rotated rx 180 ry 0 rz -180 deg; joints [-146.64, -78.365, -29.889, 64.555, 37.514, -59.043]
  Call Extruder(261.93170)
  MoveL 8303 to (238.89, 156.66, 116.27) mm, rotated rx 180 ry 0 rz 180 deg; joints [-146.617, -78.375, -29.87, 64.587, 37.531, -59.073]
  MoveL 8304 to (238.89, 156.66, 116.27) mm, rotated rx 180 ry 0 rz 180 deg; joints [-146.617, -78.375, -29.87, 64.587, 37.531, -59.073]
  Call Extruder(262.11373)
  MoveL 8305 to (238.75, 156.94, 116.27) mm, rotated rx -180 ry 0 rz 180 deg; joints [-146.589, -78.382, -29.857, 64.618, 37.552, -59.102]
  MoveL 8306 to (238.75, 156.94, 116.27) mm, rotated rx -180 ry 0 rz 180 deg; joints [-146.589, -78.382, -29.857, 64.618, 37.552, -59.102]
  Call Extruder(262.32029)
  MoveL 8307 to (238.57, 157.25, 116.27) mm, rotated rx 180 ry 0 rz 180 deg; joints [-146.557, -78.386, -29.848, 64.65, 37.577, -59.129]
  MoveL 8308 to (238.57, 157.25, 116.27) mm, rotated rx 180 ry 0 rz 180 deg; joints [-146.557, -78.386, -29.848, 64.65, 37.577, -59.129]
  Call Extruder(262.52763)
  MoveL 8309 to (238.4, 157.55, 116.27) mm, rotated rx 180 ry 0 rz 180 deg; joints [-146.526, -78.39, -29.839, 64.681, 37.602, -59.157]
  MoveL 8310 to (238.4, 157.55, 116.27) mm, rotated rx 180 ry 0 rz 180 deg; joints [-146.526, -78.39, -29.839, 64.681, 37.602, -59.157]
  Call Extruder(262.73575)
  MoveL 8311 to (238.22, 157.85, 116.27) mm, rotated rx -180 ry 0 rz 180 deg; joints [-146.495, -78.395, -29.831, 64.712, 37.627, -59.184]
  MoveL 8312 to (238.22, 157.85, 116.27) mm, rotated rx -180 ry 0 rz 180 deg; joints [-146.495, -78.395, -29.831, 64.712, 37.627, -59.184]
  Call Extruder(262.85347)
  MoveL 8313 to (238.12, 158.03, 116.27) mm, rotated rx 180 ry 0 rz 180 deg; joints [-146.477, -78.397, -29.826, 64.73, 37.641, -59.199]
  MoveL 8314 to (238.12, 158.03, 116.27) mm, rotated rx 180 ry 0 rz 180 deg; joints [-146.477, -78.397, -29.826, 64.73, 37.641, -59.199]
  Call Extruder(263.18629)
  MoveL 8315 to (237.79, 158.48, 116.27) mm, rotated rx -180 ry 0 rz 180 deg; joints [-146.427, -78.392, -29.836, 64.766, 37.686, -59.225]
  MoveL 8316 to (237.79, 158.48, 116.27) mm, rotated rx -180 ry 0 rz 180 deg; joints [-146.427, -78.392, -29.836, 64.766, 37.686, -59.225]
  Call Extruder(263.52029)
  MoveL 8317 to (237.47, 158.93, 116.27) mm, rotated rx -180 ry 0 rz 180 deg; joints [-146.377, -78.387, -29.846, 64.802, 37.731, -59.251]
  MoveL 8318 to (237.47, 158.93, 116.27) mm, rotated rx -180 ry 0 rz 180 deg; joints [-146.377, -78.387, -29.846, 64.802, 37.731, -59.251]
  Call Extruder(263.68786)
  MoveL 8319 to (237.3, 159.15, 116.27) mm, rotated rx -180 ry 0 rz 180 deg; joints [-146.352, -78.385, -29.85, 64.821, 37.754, -59.264]
  Call Extruder(264.51719)
  MoveL 8320 to (236.39, 160.19, 116.27) mm, rotated rx 180 ry 0 rz 180 deg; joints [-146.229, -78.348, -29.923, 64.88, 37.875, -59.291]
  Call Extruder(265.14825)
  MoveL 8321 to (235.6, 160.89, 116.27) mm, rotated rx 180 ry 0 rz -180 deg; joints [-146.138, -78.296, -30.029, 64.894, 37.976, -59.273]
  MoveL 8322 to (235.6, 160.89, 116.27) mm, rotated rx 180 ry 0 rz -180 deg; joints [-146.138, -78.296, -30.029, 64.894, 37.976, -59.273]
  Call Extruder(265.34587)
  MoveL 8323 to (235.35, 161.1, 116.27) mm, rotated rx 180 ry 0 rz 180 deg; joints [-146.109, -78.278, -30.065, 64.897, 38.008, -59.265]
  Call Extruder(265.67988)
  MoveL 8324 to (234.9, 161.43, 116.27) mm, rotated rx -180 ry 0 rz 180 deg; joints [-146.062, -78.24, -30.141, 64.892, 38.065, -59.239]
  MoveL 8325 to (234.9, 161.43, 116.27) mm, rotated rx -180 ry 0 rz 180 deg; joints [-146.062, -78.24, -30.141, 64.892, 38.065, -59.239]
  Call Extruder(266.01272)
  MoveL 8326 to (234.45, 161.76, 116.27) mm, rotated rx -180 ry 0 rz -180 deg; joints [-146.015, -78.202, -30.217, 64.887, 38.121, -59.214]
  MoveL 8327 to (234.45, 161.76, 116.27) mm, rotated rx -180 ry 0 rz -180 deg; joints [-146.015, -78.202, -30.217, 64.887, 38.121, -59.214]
  Call Extruder(266.19191)
  MoveL 8328 to (234.21, 161.94, 116.27) mm, rotated rx -180 ry 0 rz 180 deg; joints [-145.99, -78.181, -30.259, 64.884, 38.152, -59.2]
  MoveL 8329 to (234.21, 161.94, 116.27) mm, rotated rx -180 ry 0 rz 180 deg; joints [-145.99, -78.181, -30.259, 64.884, 38.152, -59.2]
  Call Extruder(266.40003)
  MoveL 8330 to (233.9, 162.11, 116.27) mm, rotated rx -180 ry 0 rz 180 deg; joints [-145.961, -78.151, -30.32, 64.873, 38.189, -59.174]
  MoveL 8331 to (233.9, 162.11, 116.27) mm, rotated rx -180 ry 0 rz 180 deg; joints [-145.961, -78.151, -30.32, 64.873, 38.189, -59.174]
  Call Extruder(266.60737)
  MoveL 8332 to (233.6, 162.29, 116.27) mm, rotated rx 180 ry 0 rz 180 deg; joints [-145.933, -78.12, -30.381, 64.861, 38.226, -59.148]
  MoveL 8333 to (233.6, 162.29, 116.27) mm, rotated rx 180 ry 0 rz 180 deg; joints [-145.933, -78.12, -30.381, 64.861, 38.226, -59.148]
  Call Extruder(266.81392)
  MoveL 8334 to (233.29, 162.46, 116.27) mm, rotated rx -180 ry 0 rz 180 deg; joints [-145.905, -78.09, -30.441, 64.85, 38.264, -59.122]
  MoveL 8335 to (233.29, 162.46, 116.27) mm, rotated rx -180 ry 0 rz 180 deg; joints [-145.905, -78.09, -30.441, 64.85, 38.264, -59.122]
  Call Extruder(267.01970)
  MoveL 8336 to (232.99, 162.64, 116.27) mm, rotated rx -180 ry 0 rz 180 deg; joints [-145.876, -78.06, -30.502, 64.838, 38.301, -59.096]
  MoveL 8337 to (232.99, 162.64, 116.27) mm, rotated rx -180 ry 0 rz 180 deg; joints [-145.876, -78.06, -30.502, 64.838, 38.301, -59.096]
  Call Extruder(267.17798)
  MoveL 8338 to (232.74, 162.74, 116.27) mm, rotated rx -180 ry 0 rz -180 deg; joints [-145.856, -78.031, -30.56, 64.822, 38.331, -59.067]
  MoveL 8339 to (232.74, 162.74, 116.27) mm, rotated rx -180 ry 0 rz -180 deg; joints [-145.856, -78.031, -30.56, 64.822, 38.331, -59.067]
  Call Extruder(267.33565)
  MoveL 8340 to (232.49, 162.85, 116.27) mm, rotated rx -180 ry 0 rz 180 deg; joints [-145.835, -78.002, -30.618, 64.806, 38.361, -59.038]
  MoveL 8341 to (232.49, 162.85, 116.27) mm, rotated rx -180 ry 0 rz 180 deg; joints [-145.835, -78.002, -30.618, 64.806, 38.361, -59.038]
  Call Extruder(267.50574)
  MoveL 8342 to (232.22, 162.96, 116.27) mm, rotated rx -180 ry 0 rz 180 deg; joints [-145.813, -77.971, -30.68, 64.788, 38.393, -59.007]
  MoveL 8343 to (232.22, 162.96, 116.27) mm, rotated rx -180 ry 0 rz 180 deg; joints [-145.813, -77.971, -30.68, 64.788, 38.393, -59.007]
  Call Extruder(267.68811)
  MoveL 8344 to (231.93, 163.09, 116.27) mm, rotated rx 180 ry 0 rz 180 deg; joints [-145.789, -77.937, -30.749, 64.769, 38.428, -58.972]
  MoveL 8345 to (231.93, 163.09, 116.27) mm, rotated rx 180 ry 0 rz 180 deg; joints [-145.789, -77.937, -30.749, 64.769, 38.428, -58.972]
  Call Extruder(267.86971)
  MoveL 8346 to (231.64, 163.21, 116.27) mm, rotated rx -180 ry 0 rz 180 deg; joints [-145.766, -77.903, -30.817, 64.75, 38.463, -58.938]
  MoveL 8347 to (231.64, 163.21, 116.27) mm, rotated rx -180 ry 0 rz 180 deg; joints [-145.766, -77.903, -30.817, 64.75, 38.463, -58.938]
  Call Extruder(267.98315)
  MoveL 8348 to (231.45, 163.27, 116.27) mm, rotated rx 180 ry 0 rz -180 deg; joints [-145.751, -77.879, -30.864, 64.734, 38.485, -58.912]
  MoveL 8349 to (231.45, 163.27, 116.27) mm, rotated rx 180 ry 0 rz -180 deg; joints [-145.751, -77.879, -30.864, 64.734, 38.485, -58.912]
  Call Extruder(268.09615)
  MoveL 8350 to (231.26, 163.33, 116.27) mm, rotated rx 180 ry 0 rz 180 deg; joints [-145.737, -77.856, -30.912, 64.719, 38.508, -58.887]
  MoveL 8351 to (231.26, 163.33, 116.27) mm, rotated rx 180 ry 0 rz 180 deg; joints [-145.737, -77.856, -30.912, 64.719, 38.508, -58.887]
  Call Extruder(268.20871)
  MoveL 8352 to (231.07, 163.39, 116.27) mm, rotated rx -180 ry 0 rz 180 deg; joints [-145.723, -77.832, -30.959, 64.704, 38.53, -58.862]
  MoveL 8353 to (231.07, 163.39, 116.27) mm, rotated rx -180 ry 0 rz 180 deg; joints [-145.723, -77.832, -30.959, 64.704, 38.53, -58.862]
  Call Extruder(268.32082)
  MoveL 8354 to (230.88, 163.45, 116.27) mm, rotated rx 180 ry 0 rz 180 deg; joints [-145.709, -77.808, -31.007, 64.688, 38.552, -58.836]
  MoveL 8355 to (230.88, 163.45, 116.27) mm, rotated rx 180 ry 0 rz 180 deg; joints [-145.709, -77.808, -31.007, 64.688, 38.552, -58.836]
  Call Extruder(268.43249)
  MoveL 8356 to (230.69, 163.51, 116.27) mm, rotated rx 180 ry 0 rz -180 deg; joints [-145.695, -77.785, -31.054, 64.673, 38.574, -58.811]
  MoveL 8357 to (230.69, 163.51, 116.27) mm, rotated rx 180 ry 0 rz -180 deg; joints [-145.695, -77.785, -31.054, 64.673, 38.574, -58.811]
  Call Extruder(268.56358)
  MoveL 8358 to (230.47, 163.58, 116.27) mm, rotated rx 180 ry 0 rz 180 deg; joints [-145.679, -77.756, -31.111, 64.654, 38.601, -58.78]
  MoveL 8359 to (230.47, 163.58, 116.27) mm, rotated rx 180 ry 0 rz 180 deg; joints [-145.679, -77.756, -31.111, 64.654, 38.601, -58.78]
  Call Extruder(268.69411)
  MoveL 8360 to (230.25, 163.65, 116.27) mm, rotated rx 180 ry 0 rz 180 deg; joints [-145.662, -77.728, -31.168, 64.635, 38.627, -58.749]
  MoveL 8361 to (230.25, 163.65, 116.27) mm, rotated rx 180 ry 0 rz 180 deg; joints [-145.662, -77.728, -31.168, 64.635, 38.627, -58.749]
  Call Extruder(268.82408)
  MoveL 8362 to (230.02, 163.72, 116.27) mm, rotated rx 180 ry 0 rz 180 deg; joints [-145.646, -77.699, -31.225, 64.617, 38.653, -58.719]
  MoveL 8363 to (230.02, 163.72, 116.27) mm, rotated rx 180 ry 0 rz 180 deg; joints [-145.646, -77.699, -31.225, 64.617, 38.653, -58.719]
  Call Extruder(268.95347)
  MoveL 8364 to (229.8, 163.78, 116.27) mm, rotated rx 180 ry 0 rz 180 deg; joints [-145.629, -77.671, -31.282, 64.598, 38.68, -58.688]
  MoveL 8365 to (229.8, 163.78, 116.27) mm, rotated rx 180 ry 0 rz 180 deg; joints [-145.629, -77.671, -31.282, 64.598, 38.68, -58.688]
  Call Extruder(269.07545)
  MoveL 8366 to (229.59, 163.84, 116.27) mm, rotated rx 180 ry 0 rz -180 deg; joints [-145.614, -77.643, -31.338, 64.579, 38.705, -58.657]
  MoveL 8367 to (229.59, 163.84, 116.27) mm, rotated rx 180 ry 0 rz -180 deg; joints [-145.614, -77.643, -31.338, 64.579, 38.705, -58.657]
  Call Extruder(269.19030)
  MoveL 8368 to (229.38, 163.88, 116.27) mm, rotated rx 180 ry 0 rz -180 deg; joints [-145.601, -77.615, -31.394, 64.559, 38.728, -58.625]
  MoveL 8369 to (229.38, 163.88, 116.27) mm, rotated rx 180 ry 0 rz -180 deg; joints [-145.601, -77.615, -31.394, 64.559, 38.728, -58.625]
  Call Extruder(269.30469)
  MoveL 8370 to (229.18, 163.93, 116.27) mm, rotated rx 180 ry 0 rz -180 deg; joints [-145.587, -77.588, -31.449, 64.539, 38.752, -58.594]
  MoveL 8371 to (229.18, 163.93, 116.27) mm, rotated rx 180 ry 0 rz -180 deg; joints [-145.587, -77.588, -31.449, 64.539, 38.752, -58.594]
  Call Extruder(269.41863)
  MoveL 8372 to (228.97, 163.97, 116.27) mm, rotated rx 180 ry 0 rz 180 deg; joints [-145.573, -77.56, -31.505, 64.519, 38.776, -58.563]
  MoveL 8373 to (228.97, 163.97, 116.27) mm, rotated rx 180 ry 0 rz 180 deg; joints [-145.573, -77.56, -31.505, 64.519, 38.776, -58.563]
  Call Extruder(269.53212)
  MoveL 8374 to (228.77, 164.02, 116.27) mm, rotated rx 180 ry 0 rz 180 deg; joints [-145.559, -77.533, -31.56, 64.499, 38.799, -58.532]
  MoveL 8375 to (228.77, 164.02, 116.27) mm, rotated rx 180 ry 0 rz 180 deg; joints [-145.559, -77.533, -31.56, 64.499, 38.799, -58.532]
  Call Extruder(269.66941)
  MoveL 8376 to (228.52, 164.07, 116.27) mm, rotated rx -180 ry 0 rz -180 deg; joints [-145.543, -77.499, -31.628, 64.475, 38.828, -58.493]
  MoveL 8377 to (228.52, 164.07, 116.27) mm, rotated rx -180 ry 0 rz -180 deg; joints [-145.543, -77.499, -31.628, 64.475, 38.828, -58.493]
  Call Extruder(269.80608)
  MoveL 8378 to (228.27, 164.12, 116.27) mm, rotated rx -180 ry 0 rz -180 deg; joints [-145.527, -77.465, -31.697, 64.45, 38.857, -58.454]
  MoveL 8379 to (228.27, 164.12, 116.27) mm, rotated rx -180 ry 0 rz -180 deg; joints [-145.527, -77.465, -31.697, 64.45, 38.857, -58.454]
  Call Extruder(269.94214)
  MoveL 8380 to (228.02, 164.17, 116.27) mm, rotated rx -180 ry 0 rz -180 deg; joints [-145.51, -77.431, -31.765, 64.425, 38.886, -58.416]
  MoveL 8381 to (228.02, 164.17, 116.27) mm, rotated rx -180 ry 0 rz -180 deg; joints [-145.51, -77.431, -31.765, 64.425, 38.886, -58.416]
  Call Extruder(270.07759)
  MoveL 8382 to (227.77, 164.22, 116.27) mm, rotated rx 180 ry 0 rz -180 deg; joints [-145.494, -77.397, -31.833, 64.401, 38.914, -58.377]
  MoveL 8383 to (227.77, 164.22, 116.27) mm, rotated rx 180 ry 0 rz -180 deg; joints [-145.494, -77.397, -31.833, 64.401, 38.914, -58.377]
  Call Extruder(270.21244)
  MoveL 8384 to (227.52, 164.27, 116.27) mm, rotated rx 180 ry 0 rz 180 deg; joints [-145.477, -77.363, -31.901, 64.376, 38.943, -58.339]
  MoveL 8385 to (227.52, 164.27, 116.27) mm, rotated rx 180 ry 0 rz 180 deg; joints [-145.477, -77.363, -31.901, 64.376, 38.943, -58.339]
  Call Extruder(270.34667)
  MoveL 8386 to (227.27, 164.32, 116.27) mm, rotated rx 180 ry 0 rz -180 deg; joints [-145.461, -77.329, -31.968, 64.352, 38.972, -58.301]
  MoveL 8387 to (227.27, 164.32, 116.27) mm, rotated rx 180 ry 0 rz -180 deg; joints [-145.461, -77.329, -31.968, 64.352, 38.972, -58.301]
  Call Extruder(270.48029)
  MoveL 8388 to (227.03, 164.37, 116.27) mm, rotated rx -180 ry 0 rz -180 deg; joints [-145.444, -77.296, -32.036, 64.328, 39.001, -58.263]
  MoveL 8389 to (227.03, 164.37, 116.27) mm, rotated rx -180 ry 0 rz -180 deg; joints [-145.444, -77.296, -32.036, 64.328, 39.001, -58.263]
  Call Extruder(270.64240)
  MoveL 8390 to (226.72, 164.41, 116.27) mm, rotated rx 180 ry 0 rz 180 deg; joints [-145.425, -77.253, -32.122, 64.296, 39.036, -58.214]
  MoveL 8391 to (226.72, 164.41, 116.27) mm, rotated rx 180 ry 0 rz 180 deg; joints [-145.425, -77.253, -32.122, 64.296, 39.036, -58.214]
  Call Extruder(270.80377)
  MoveL 8392 to (226.41, 164.46, 116.27) mm, rotated rx 180 ry 0 rz -180 deg; joints [-145.406, -77.211, -32.207, 64.265, 39.071, -58.165]
  MoveL 8393 to (226.41, 164.46, 116.27) mm, rotated rx 180 ry 0 rz -180 deg; joints [-145.406, -77.211, -32.207, 64.265, 39.071, -58.165]
  Call Extruder(270.96442)
  MoveL 8394 to (226.11, 164.51, 116.27) mm, rotated rx 180 ry 0 rz -180 deg; joints [-145.386, -77.168, -32.292, 64.234, 39.106, -58.117]
  MoveL 8395 to (226.11, 164.51, 116.27) mm, rotated rx 180 ry 0 rz -180 deg; joints [-145.386, -77.168, -32.292, 64.234, 39.106, -58.117]
  Call Extruder(271.12435)
  MoveL 8396 to (225.8, 164.56, 116.27) mm, rotated rx -180 ry 0 rz 180 deg; joints [-145.367, -77.126, -32.377, 64.202, 39.141, -58.068]
  MoveL 8397 to (225.8, 164.56, 116.27) mm, rotated rx -180 ry 0 rz 180 deg; joints [-145.367, -77.126, -32.377, 64.202, 39.141, -58.068]
  Call Extruder(271.28354)
  MoveL 8398 to (225.5, 164.61, 116.27) mm, rotated rx 180 ry 0 rz -180 deg; joints [-145.348, -77.084, -32.462, 64.172, 39.176, -58.02]
  MoveL 8399 to (225.5, 164.61, 116.27) mm, rotated rx 180 ry 0 rz -180 deg; joints [-145.348, -77.084, -32.462, 64.172, 39.176, -58.02]
  Call Extruder(271.44201)
  MoveL 8400 to (225.19, 164.66, 116.27) mm, rotated rx -180 ry 0 rz 180 deg; joints [-145.328, -77.042, -32.547, 64.141, 39.211, -57.972]
  MoveL 8401 to (225.19, 164.66, 116.27) mm, rotated rx -180 ry 0 rz 180 deg; joints [-145.328, -77.042, -32.547, 64.141, 39.211, -57.972]
  Call Extruder(271.64088)
  MoveL 8402 to (224.8, 164.7, 116.27) mm, rotated rx 180 ry 0 rz 180 deg; joints [-145.305, -76.987, -32.657, 64.099, 39.255, -57.908]
  MoveL 8403 to (224.8, 164.7, 116.27) mm, rotated rx 180 ry 0 rz 180 deg; joints [-145.305, -76.987, -32.657, 64.099, 39.255, -57.908]
  Call Extruder(271.83889)
  MoveL 8404 to (224.42, 164.75, 116.27) mm, rotated rx 180 ry 0 rz 180 deg; joints [-145.281, -76.932, -32.767, 64.058, 39.299, -57.844]
  MoveL 8405 to (224.42, 164.75, 116.27) mm, rotated rx 180 ry 0 rz 180 deg; joints [-145.281, -76.932, -32.767, 64.058, 39.299, -57.844]
  Call Extruder(272.03603)
  MoveL 8406 to (224.03, 164.79, 116.27) mm, rotated rx -180 ry 0 rz 180 deg; joints [-145.258, -76.878, -32.877, 64.017, 39.343, -57.781]
  MoveL 8407 to (224.03, 164.79, 116.27) mm, rotated rx -180 ry 0 rz 180 deg; joints [-145.258, -76.878, -32.877, 64.017, 39.343, -57.781]
  Call Extruder(272.23230)
  MoveL 8408 to (223.64, 164.84, 116.27) mm, rotated rx 180 ry 0 rz 180 deg; joints [-145.234, -76.823, -32.987, 63.976, 39.387, -57.718]
  MoveL 8409 to (223.64, 164.84, 116.27) mm, rotated rx 180 ry 0 rz 180 deg; joints [-145.234, -76.823, -32.987, 63.976, 39.387, -57.718]
  Call Extruder(272.47797)
  MoveL 8410 to (223.15, 164.89, 116.27) mm, rotated rx 180 ry 0 rz -180 deg; joints [-145.206, -76.754, -33.127, 63.923, 39.442, -57.637]
  MoveL 8411 to (223.15, 164.89, 116.27) mm, rotated rx 180 ry 0 rz -180 deg; joints [-145.206, -76.754, -33.127, 63.923, 39.442, -57.637]
  Call Extruder(272.77266)
  MoveL 8412 to (222.56, 164.93, 116.27) mm, rotated rx -180 ry 0 rz 180 deg; joints [-145.172, -76.669, -33.298, 63.858, 39.509, -57.538]
  MoveL 8413 to (222.56, 164.93, 116.27) mm, rotated rx -180 ry 0 rz 180 deg; joints [-145.172, -76.669, -33.298, 63.858, 39.509, -57.538]
  Call Extruder(273.06601)
  MoveL 8414 to (221.97, 164.98, 116.27) mm, rotated rx 180 ry 0 rz 180 deg; joints [-145.138, -76.585, -33.467, 63.794, 39.575, -57.44]
  MoveL 8415 to (221.97, 164.98, 116.27) mm, rotated rx 180 ry 0 rz 180 deg; joints [-145.138, -76.585, -33.467, 63.794, 39.575, -57.44]
  Call Extruder(273.49932)
  MoveL 8416 to (221.1, 165.02, 116.27) mm, rotated rx 180 ry 0 rz 180 deg; joints [-145.088, -76.458, -33.723, 63.696, 39.674, -57.291]
  MoveL 8417 to (221.1, 165.02, 116.27) mm, rotated rx 180 ry 0 rz 180 deg; joints [-145.088, -76.458, -33.723, 63.696, 39.674, -57.291]
  Call Extruder(274.07148)
  MoveL 8418 to (219.94, 165.07, 116.27) mm, rotated rx -180 ry 0 rz -180 deg; joints [-145.024, -76.289, -34.063, 63.565, 39.804, -57.092]
  MoveL 8419 to (219.94, 165.07, 116.27) mm, rotated rx -180 ry 0 rz -180 deg; joints [-145.024, -76.289, -34.063, 63.565, 39.804, -57.092]
  Call Extruder(274.49936)
  MoveL 8420 to (219.06, 165.09, 116.27) mm, rotated rx 180 ry 0 rz 180 deg; joints [-144.977, -76.161, -34.321, 63.466, 39.901, -56.941]
  Call Extruder(391.14801)
  MoveL 8421 to (-19.06, 165.09, 116.27) mm, rotated rx 180 ry 0 rz 180 deg; joints [-127.435, -55.313, -78.779, 61.958, 64.114, -39.339]
  MoveL 8422 to (-19.06, 165.09, 116.27) mm, rotated rx 180 ry 0 rz 180 deg; joints [-127.435, -55.313, -78.779, 61.958, 64.114, -39.339]
  Call Extruder(391.86364)
  MoveL 8423 to (-20.52, 165.05, 116.27) mm, rotated rx 180 ry 0 rz 180 deg; joints [-127.291, -55.234, -78.962, 62.037, 64.254, -39.291]
  MoveL 8424 to (-20.52, 165.05, 116.27) mm, rotated rx 180 ry 0 rz 180 deg; joints [-127.291, -55.234, -78.962, 62.037, 64.254, -39.291]
  Call Extruder(392.43838)
  MoveL 8425 to (-21.68, 165, 116.27) mm, rotated rx -180 ry 0 rz 180 deg; joints [-127.178, -55.171, -79.109, 62.099, 64.365, -39.251]
  MoveL 8426 to (-21.68, 165, 116.27) mm, rotated rx -180 ry 0 rz 180 deg; joints [-127.178, -55.171, -79.109, 62.099, 64.365, -39.251]
  Call Extruder(392.73174)
  MoveL 8427 to (-22.27, 164.95, 116.27) mm, rotated rx -180 ry 0 rz 180 deg; joints [-127.122, -55.137, -79.188, 62.128, 64.422, -39.228]
  MoveL 8428 to (-22.27, 164.95, 116.27) mm, rotated rx -180 ry 0 rz 180 deg; joints [-127.122, -55.137, -79.188, 62.128, 64.422, -39.228]
  Call Extruder(393.02643)
  MoveL 8429 to (-22.86, 164.91, 116.27) mm, rotated rx 180 ry 0 rz 180 deg; joints [-127.065, -55.103, -79.266, 62.157, 64.478, -39.205]
  MoveL 8430 to (-22.86, 164.91, 116.27) mm, rotated rx 180 ry 0 rz 180 deg; joints [-127.065, -55.103, -79.266, 62.157, 64.478, -39.205]
  Call Extruder(393.32246)
  MoveL 8431 to (-23.45, 164.86, 116.27) mm, rotated rx -180 ry 0 rz 180 deg; joints [-127.009, -55.07, -79.344, 62.187, 64.534, -39.182]
  MoveL 8432 to (-23.45, 164.86, 116.27) mm, rotated rx -180 ry 0 rz 180 deg; joints [-127.009, -55.07, -79.344, 62.187, 64.534, -39.182]
  Call Extruder(393.51873)
  MoveL 8433 to (-23.83, 164.82, 116.27) mm, rotated rx 180 ry 0 rz 180 deg; joints [-126.973, -55.046, -79.397, 62.205, 64.571, -39.166]
  MoveL 8434 to (-23.83, 164.82, 116.27) mm, rotated rx 180 ry 0 rz 180 deg; joints [-126.973, -55.046, -79.397, 62.205, 64.571, -39.166]
  Call Extruder(393.71587)
  MoveL 8435 to (-24.22, 164.77, 116.27) mm, rotated rx 180 ry 0 rz 180 deg; joints [-126.937, -55.023, -79.451, 62.223, 64.608, -39.149]
  MoveL 8436 to (-24.22, 164.77, 116.27) mm, rotated rx 180 ry 0 rz 180 deg; joints [-126.937, -55.023, -79.451, 62.223, 64.608, -39.149]
  Call Extruder(393.91388)
  MoveL 8437 to (-24.61, 164.72, 116.27) mm, rotated rx -180 ry 0 rz 180 deg; joints [-126.901, -55, -79.505, 62.241, 64.645, -39.132]
  MoveL 8438 to (-24.61, 164.72, 116.27) mm, rotated rx -180 ry 0 rz 180 deg; joints [-126.901, -55, -79.505, 62.241, 64.645, -39.132]
  Call Extruder(394.11275)
  MoveL 8439 to (-25, 164.68, 116.27) mm, rotated rx 180 ry 0 rz 180 deg; joints [-126.865, -54.977, -79.558, 62.259, 64.682, -39.116]
  MoveL 8440 to (-25, 164.68, 116.27) mm, rotated rx 180 ry 0 rz 180 deg; joints [-126.865, -54.977, -79.558, 62.259, 64.682, -39.116]
  Call Extruder(394.29183)
  MoveL 8441 to (-25.34, 164.63, 116.27) mm, rotated rx 180 ry 0 rz 180 deg; joints [-126.834, -54.956, -79.607, 62.275, 64.715, -39.1]
  MoveL 8442 to (-25.34, 164.63, 116.27) mm, rotated rx 180 ry 0 rz 180 deg; joints [-126.834, -54.956, -79.607, 62.275, 64.715, -39.1]
  Call Extruder(394.45103)
  MoveL 8443 to (-25.65, 164.58, 116.27) mm, rotated rx 180 ry 0 rz 180 deg; joints [-126.806, -54.937, -79.651, 62.288, 64.744, -39.085]
  MoveL 8444 to (-25.65, 164.58, 116.27) mm, rotated rx 180 ry 0 rz 180 deg; joints [-126.806, -54.937, -79.651, 62.288, 64.744, -39.085]
  Call Extruder(394.61095)
  MoveL 8445 to (-25.96, 164.53, 116.27) mm, rotated rx -180 ry 0 rz 180 deg; joints [-126.779, -54.918, -79.695, 62.301, 64.773, -39.071]
  MoveL 8446 to (-25.96, 164.53, 116.27) mm, rotated rx -180 ry 0 rz 180 deg; joints [-126.779, -54.918, -79.695, 62.301, 64.773, -39.071]
  Call Extruder(394.77161)
  MoveL 8447 to (-26.26, 164.49, 116.27) mm, rotated rx 180 ry 0 rz 180 deg; joints [-126.751, -54.9, -79.739, 62.314, 64.802, -39.057]
  MoveL 8448 to (-26.26, 164.49, 116.27) mm, rotated rx 180 ry 0 rz 180 deg; joints [-126.751, -54.9, -79.739, 62.314, 64.802, -39.057]
  Call Extruder(394.93299)
  MoveL 8449 to (-26.57, 164.44, 116.27) mm, rotated rx 180 ry 0 rz 180 deg; joints [-126.723, -54.881, -79.783, 62.327, 64.831, -39.042]
  MoveL 8450 to (-26.57, 164.44, 116.27) mm, rotated rx 180 ry 0 rz 180 deg; joints [-126.723, -54.881, -79.783, 62.327, 64.831, -39.042]
  Call Extruder(395.09509)
  MoveL 8451 to (-26.87, 164.39, 116.27) mm, rotated rx -180 ry 0 rz 180 deg; joints [-126.696, -54.862, -79.827, 62.341, 64.86, -39.028]
  MoveL 8452 to (-26.87, 164.39, 116.27) mm, rotated rx -180 ry 0 rz 180 deg; joints [-126.696, -54.862, -79.827, 62.341, 64.86, -39.028]
  Call Extruder(395.24330)
  MoveL 8453 to (-27.15, 164.34, 116.27) mm, rotated rx 180 ry 0 rz 180 deg; joints [-126.671, -54.844, -79.867, 62.352, 64.886, -39.014]
  MoveL 8454 to (-27.15, 164.34, 116.27) mm, rotated rx 180 ry 0 rz 180 deg; joints [-126.671, -54.844, -79.867, 62.352, 64.886, -39.014]
  Call Extruder(395.37753)
  MoveL 8455 to (-27.4, 164.29, 116.27) mm, rotated rx 180 ry 0 rz -180 deg; joints [-126.649, -54.828, -79.905, 62.362, 64.91, -39.001]
  MoveL 8456 to (-27.4, 164.29, 116.27) mm, rotated rx 180 ry 0 rz -180 deg; joints [-126.649, -54.828, -79.905, 62.362, 64.91, -39.001]
  Call Extruder(395.51237)
  MoveL 8457 to (-27.65, 164.24, 116.27) mm, rotated rx 180 ry 0 rz 180 deg; joints [-126.628, -54.812, -79.942, 62.372, 64.933, -38.988]
  MoveL 8458 to (-27.65, 164.24, 116.27) mm, rotated rx 180 ry 0 rz 180 deg; joints [-126.628, -54.812, -79.942, 62.372, 64.933, -38.988]
  Call Extruder(395.64782)
  MoveL 8459 to (-27.9, 164.19, 116.27) mm, rotated rx 180 ry 0 rz 180 deg; joints [-126.606, -54.796, -79.979, 62.382, 64.957, -38.975]
  MoveL 8460 to (-27.9, 164.19, 116.27) mm, rotated rx 180 ry 0 rz 180 deg; joints [-126.606, -54.796, -79.979, 62.382, 64.957, -38.975]
  Call Extruder(395.78388)
  MoveL 8461 to (-28.15, 164.14, 116.27) mm, rotated rx -180 ry 0 rz 180 deg; joints [-126.584, -54.78, -80.016, 62.392, 64.98, -38.962]
  MoveL 8462 to (-28.15, 164.14, 116.27) mm, rotated rx -180 ry 0 rz 180 deg; joints [-126.584, -54.78, -80.016, 62.392, 64.98, -38.962]
  Call Extruder(395.92056)
  MoveL 8463 to (-28.4, 164.09, 116.27) mm, rotated rx -180 ry 0 rz 180 deg; joints [-126.562, -54.764, -80.054, 62.402, 65.004, -38.95]
  MoveL 8464 to (-28.4, 164.09, 116.27) mm, rotated rx -180 ry 0 rz 180 deg; joints [-126.562, -54.764, -80.054, 62.402, 65.004, -38.95]
  Call Extruder(396.05784)
  MoveL 8465 to (-28.65, 164.04, 116.27) mm, rotated rx -180 ry 0 rz 180 deg; joints [-126.54, -54.748, -80.091, 62.412, 65.028, -38.937]
  MoveL 8466 to (-28.65, 164.04, 116.27) mm, rotated rx -180 ry 0 rz 180 deg; joints [-126.54, -54.748, -80.091, 62.412, 65.028, -38.937]
  Call Extruder(396.18351)
  MoveL 8467 to (-28.87, 164, 116.27) mm, rotated rx 180 ry 0 rz 180 deg; joints [-126.52, -54.734, -80.125, 62.421, 65.049, -38.925]
  MoveL 8468 to (-28.87, 164, 116.27) mm, rotated rx 180 ry 0 rz 180 deg; joints [-126.52, -54.734, -80.125, 62.421, 65.049, -38.925]
  Call Extruder(396.29745)
  MoveL 8469 to (-29.08, 163.95, 116.27) mm, rotated rx -180 ry 0 rz 180 deg; joints [-126.503, -54.72, -80.156, 62.428, 65.068, -38.914]
  MoveL 8470 to (-29.08, 163.95, 116.27) mm, rotated rx -180 ry 0 rz 180 deg; joints [-126.503, -54.72, -80.156, 62.428, 65.068, -38.914]
  Call Extruder(396.41184)
  MoveL 8471 to (-29.28, 163.91, 116.27) mm, rotated rx 180 ry 0 rz 180 deg; joints [-126.485, -54.707, -80.187, 62.436, 65.088, -38.903]
  MoveL 8472 to (-29.28, 163.91, 116.27) mm, rotated rx 180 ry 0 rz 180 deg; joints [-126.485, -54.707, -80.187, 62.436, 65.088, -38.903]
  Call Extruder(396.52669)
  MoveL 8473 to (-29.48, 163.86, 116.27) mm, rotated rx -180 ry 0 rz -180 deg; joints [-126.467, -54.694, -80.218, 62.444, 65.107, -38.892]
  MoveL 8474 to (-29.48, 163.86, 116.27) mm, rotated rx -180 ry 0 rz -180 deg; joints [-126.467, -54.694, -80.218, 62.444, 65.107, -38.892]
  Call Extruder(396.64199)
  MoveL 8475 to (-29.69, 163.82, 116.27) mm, rotated rx -180 ry 0 rz 180 deg; joints [-126.45, -54.681, -80.249, 62.452, 65.126, -38.881]
  MoveL 8476 to (-29.69, 163.82, 116.27) mm, rotated rx -180 ry 0 rz 180 deg; joints [-126.45, -54.681, -80.249, 62.452, 65.126, -38.881]
  Call Extruder(396.77138)
  MoveL 8477 to (-29.91, 163.75, 116.27) mm, rotated rx 180 ry 0 rz 180 deg; joints [-126.432, -54.665, -80.286, 62.459, 65.147, -38.867]
  MoveL 8478 to (-29.91, 163.75, 116.27) mm, rotated rx 180 ry 0 rz 180 deg; joints [-126.432, -54.665, -80.286, 62.459, 65.147, -38.867]
  Call Extruder(396.90134)
  MoveL 8479 to (-30.14, 163.68, 116.27) mm, rotated rx -180 ry 0 rz 180 deg; joints [-126.414, -54.649, -80.323, 62.466, 65.168, -38.853]
  MoveL 8480 to (-30.14, 163.68, 116.27) mm, rotated rx -180 ry 0 rz 180 deg; joints [-126.414, -54.649, -80.323, 62.466, 65.168, -38.853]
  Call Extruder(397.03187)
  MoveL 8481 to (-30.36, 163.61, 116.27) mm, rotated rx 180 ry 0 rz 180 deg; joints [-126.396, -54.633, -80.36, 62.472, 65.189, -38.839]
  MoveL 8482 to (-30.36, 163.61, 116.27) mm, rotated rx 180 ry 0 rz 180 deg; joints [-126.396, -54.633, -80.36, 62.472, 65.189, -38.839]
  Call Extruder(397.16296)
  MoveL 8483 to (-30.58, 163.55, 116.27) mm, rotated rx 180 ry 0 rz 180 deg; joints [-126.378, -54.617, -80.397, 62.479, 65.211, -38.824]
  MoveL 8484 to (-30.58, 163.55, 116.27) mm, rotated rx 180 ry 0 rz 180 deg; joints [-126.378, -54.617, -80.397, 62.479, 65.211, -38.824]
  Call Extruder(397.28461)
  MoveL 8485 to (-30.79, 163.48, 116.27) mm, rotated rx -180 ry 0 rz -180 deg; joints [-126.361, -54.603, -80.431, 62.485, 65.23, -38.811]
  MoveL 8486 to (-30.79, 163.48, 116.27) mm, rotated rx -180 ry 0 rz -180 deg; joints [-126.361, -54.603, -80.431, 62.485, 65.23, -38.811]
  Call Extruder(397.39672)
  MoveL 8487 to (-30.98, 163.42, 116.27) mm, rotated rx 180 ry 0 rz 180 deg; joints [-126.347, -54.589, -80.463, 62.49, 65.248, -38.799]
  MoveL 8488 to (-30.98, 163.42, 116.27) mm, rotated rx 180 ry 0 rz 180 deg; joints [-126.347, -54.589, -80.463, 62.49, 65.248, -38.799]
  Call Extruder(397.50928)
  MoveL 8489 to (-31.17, 163.36, 116.27) mm, rotated rx -180 ry 0 rz 180 deg; joints [-126.332, -54.576, -80.495, 62.496, 65.265, -38.786]
  MoveL 8490 to (-31.17, 163.36, 116.27) mm, rotated rx -180 ry 0 rz 180 deg; joints [-126.332, -54.576, -80.495, 62.496, 65.265, -38.786]
  Call Extruder(397.54120)
  MoveL 8491 to (-31.22, 163.34, 116.27) mm, rotated rx 180 ry 0 rz -180 deg; joints [-126.327, -54.572, -80.504, 62.497, 65.27, -38.783]
  Set speed (130.0 mm/s)
  MoveL 8492 to (-34.34, 162.18, 116.27) mm, rotated rx 180 ry 0 rz 180 deg; joints [-126.091, -54.338, -81.05, 62.573, 65.563, -38.562]
  MoveL 8493 to (-34.34, 162.18, 125.68) mm, rotated rx -180 ry 0 rz 180 deg; joints [-126.091, -53.09, -81.528, 62.887, 65.21, -39.315]
  MoveL 8494 to (-31.64, 163.21, 125.68) mm, rotated rx 180 ry 0 rz 180 deg; joints [-126.294, -53.298, -81.052, 62.825, 64.958, -39.506]
  Set speed (30.0 mm/s)
  MoveL 8495 to (-31.64, 163.21, 125.68) mm, rotated rx 180 ry 0 rz 180 deg; joints [-126.294, -53.298, -81.052, 62.825, 64.958, -39.506]
  Call Extruder(397.72317)
  MoveL 8496 to (-31.93, 163.09, 125.68) mm, rotated rx 180 ry 0 rz 180 deg; joints [-126.273, -53.274, -81.105, 62.83, 64.985, -39.484]
  MoveL 8497 to (-31.93, 163.09, 125.68) mm, rotated rx 180 ry 0 rz 180 deg; joints [-126.273, -53.274, -81.105, 62.83, 64.985, -39.484]
  Call Extruder(397.90591)
  MoveL 8498 to (-32.22, 162.97, 125.68) mm, rotated rx 180 ry 0 rz -180 deg; joints [-126.252, -53.251, -81.158, 62.836, 65.012, -39.462]
  MoveL 8499 to (-32.22, 162.97, 125.68) mm, rotated rx 180 ry 0 rz -180 deg; joints [-126.252, -53.251, -81.158, 62.836, 65.012, -39.462]
  Call Extruder(398.07632)
  MoveL 8500 to (-32.49, 162.85, 125.68) mm, rotated rx 180 ry 0 rz 180 deg; joints [-126.233, -53.23, -81.207, 62.841, 65.037, -39.442]
  MoveL 8501 to (-32.49, 162.85, 125.68) mm, rotated rx 180 ry 0 rz 180 deg; joints [-126.233, -53.23, -81.207, 62.841, 65.037, -39.442]
  Call Extruder(398.23430)
  MoveL 8502 to (-32.74, 162.74, 125.68) mm, rotated rx 180 ry 0 rz 180 deg; joints [-126.215, -53.21, -81.253, 62.845, 65.06, -39.423]
  MoveL 8503 to (-32.74, 162.74, 125.68) mm, rotated rx 180 ry 0 rz 180 deg; joints [-126.215, -53.21, -81.253, 62.845, 65.06, -39.423]
  Call Extruder(398.39287)
  MoveL 8504 to (-32.99, 162.64, 125.68) mm, rotated rx 180 ry 0 rz 180 deg; joints [-126.197, -53.19, -81.299, 62.85, 65.083, -39.404]
  MoveL 8505 to (-32.99, 162.64, 125.68) mm, rotated rx 180 ry 0 rz 180 deg; joints [-126.197, -53.19, -81.299, 62.85, 65.083, -39.404]
  Call Extruder(398.59904)
  MoveL 8506 to (-33.29, 162.46, 125.68) mm, rotated rx -180 ry 0 rz 180 deg; joints [-126.179, -53.162, -81.362, 62.851, 65.111, -39.375]
  MoveL 8507 to (-33.29, 162.46, 125.68) mm, rotated rx -180 ry 0 rz 180 deg; joints [-126.179, -53.162, -81.362, 62.851, 65.111, -39.375]
  Call Extruder(398.80598)
  MoveL 8508 to (-33.6, 162.29, 125.68) mm, rotated rx 180 ry 0 rz 180 deg; joints [-126.16, -53.135, -81.425, 62.852, 65.139, -39.347]
  MoveL 8509 to (-33.6, 162.29, 125.68) mm, rotated rx 180 ry 0 rz 180 deg; joints [-126.16, -53.135, -81.425, 62.852, 65.139, -39.347]
  Call Extruder(399.01371)
  MoveL 8510 to (-33.9, 162.11, 125.68) mm, rotated rx 180 ry 0 rz 180 deg; joints [-126.142, -53.107, -81.488, 62.853, 65.167, -39.319]
  MoveL 8511 to (-33.9, 162.11, 125.68) mm, rotated rx 180 ry 0 rz 180 deg; joints [-126.142, -53.107, -81.488, 62.853, 65.167, -39.319]
  Call Extruder(399.22221)
  MoveL 8512 to (-34.21, 161.94, 125.68) mm, rotated rx 180 ry 0 rz 180 deg; joints [-126.123, -53.08, -81.551, 62.854, 65.195, -39.291]
  MoveL 8513 to (-34.21, 161.94, 125.68) mm, rotated rx 180 ry 0 rz 180 deg; joints [-126.123, -53.08, -81.551, 62.854, 65.195, -39.291]
  Call Extruder(399.40175)
  MoveL 8514 to (-34.45, 161.76, 125.68) mm, rotated rx -180 ry 0 rz 180 deg; joints [-126.111, -53.055, -81.608, 62.851, 65.217, -39.264]
  MoveL 8515 to (-34.45, 161.76, 125.68) mm, rotated rx -180 ry 0 rz 180 deg; joints [-126.111, -53.055, -81.608, 62.851, 65.217, -39.264]
  Call Extruder(399.73518)
  MoveL 8516 to (-34.9, 161.43, 125.68) mm, rotated rx 180 ry 0 rz 180 deg; joints [-126.089, -53.01, -81.711, 62.846, 65.258, -39.214]
  MoveL 8517 to (-34.9, 161.43, 125.68) mm, rotated rx 180 ry 0 rz 180 deg; joints [-126.089, -53.01, -81.711, 62.846, 65.258, -39.214]
  Call Extruder(400.06980)
  MoveL 8518 to (-35.35, 161.1, 125.68) mm, rotated rx 180 ry 0 rz -180 deg; joints [-126.067, -52.965, -81.815, 62.841, 65.299, -39.165]
  Call Extruder(400.89771)
  MoveL 8519 to (-36.39, 160.19, 125.68) mm, rotated rx 180 ry 0 rz 180 deg; joints [-126.027, -52.851, -82.079, 62.814, 65.392, -39.033]
  Call Extruder(401.72565)
  MoveL 8520 to (-37.3, 159.15, 125.68) mm, rotated rx 180 ry 0 rz 180 deg; joints [-126.011, -52.734, -82.347, 62.766, 65.472, -38.89]
  Call Extruder(401.89295)
  MoveL 8521 to (-37.47, 158.93, 125.68) mm, rotated rx 180 ry 0 rz 180 deg; joints [-126.011, -52.711, -82.401, 62.754, 65.486, -38.86]
  MoveL 8522 to (-37.47, 158.93, 125.68) mm, rotated rx 180 ry 0 rz 180 deg; joints [-126.011, -52.711, -82.401, 62.754, 65.486, -38.86]
  Call Extruder(402.22638)
  MoveL 8523 to (-37.79, 158.48, 125.68) mm, rotated rx 180 ry 0 rz 180 deg; joints [-126.011, -52.664, -82.51, 62.729, 65.514, -38.8]
  MoveL 8524 to (-37.79, 158.48, 125.68) mm, rotated rx 180 ry 0 rz 180 deg; joints [-126.011, -52.664, -82.51, 62.729, 65.514, -38.8]
  Call Extruder(402.55863)
  MoveL 8525 to (-38.12, 158.02, 125.68) mm, rotated rx -180 ry 0 rz -180 deg; joints [-126.011, -52.617, -82.618, 62.704, 65.542, -38.74]
  MoveL 8526 to (-38.12, 158.02, 125.68) mm, rotated rx -180 ry 0 rz -180 deg; joints [-126.011, -52.617, -82.618, 62.704, 65.542, -38.74]
  Call Extruder(402.67630)
  MoveL 8527 to (-38.22, 157.85, 125.68) mm, rotated rx 180 ry 0 rz -180 deg; joints [-126.013, -52.6, -82.656, 62.693, 65.55, -38.718]
  MoveL 8528 to (-38.22, 157.85, 125.68) mm, rotated rx 180 ry 0 rz -180 deg; joints [-126.013, -52.6, -82.656, 62.693, 65.55, -38.718]
  Call Extruder(402.88403)
  MoveL 8529 to (-38.4, 157.55, 125.68) mm, rotated rx -180 ry 0 rz 180 deg; joints [-126.018, -52.571, -82.724, 62.673, 65.565, -38.679]
  MoveL 8530 to (-38.4, 157.55, 125.68) mm, rotated rx -180 ry 0 rz 180 deg; joints [-126.018, -52.571, -82.724, 62.673, 65.565, -38.679]
  Call Extruder(403.09097)
  MoveL 8531 to (-38.57, 157.25, 125.68) mm, rotated rx 180 ry 0 rz 180 deg; joints [-126.023, -52.542, -82.792, 62.654, 65.58, -38.64]
  MoveL 8532 to (-38.57, 157.25, 125.68) mm, rotated rx 180 ry 0 rz 180 deg; joints [-126.023, -52.542, -82.792, 62.654, 65.58, -38.64]
  Call Extruder(403.29714)
  MoveL 8533 to (-38.75, 156.94, 125.68) mm, rotated rx 180 ry 0 rz -180 deg; joints [-126.028, -52.512, -82.86, 62.634, 65.594, -38.6]
  MoveL 8534 to (-38.75, 156.94, 125.68) mm, rotated rx 180 ry 0 rz -180 deg; joints [-126.028, -52.512, -82.86, 62.634, 65.594, -38.6]
  Call Extruder(403.47882)
  MoveL 8535 to (-38.89, 156.66, 125.68) mm, rotated rx 180 ry 0 rz -180 deg; joints [-126.034, -52.487, -82.919, 62.615, 65.606, -38.565]
  MoveL 8536 to (-38.89, 156.66, 125.68) mm, rotated rx 180 ry 0 rz -180 deg; joints [-126.034, -52.487, -82.919, 62.615, 65.606, -38.565]
  Call Extruder(403.63681)
  MoveL 8537 to (-39, 156.42, 125.68) mm, rotated rx 180 ry 0 rz -180 deg; joints [-126.042, -52.465, -82.97, 62.597, 65.614, -38.534]
  MoveL 8538 to (-39, 156.42, 125.68) mm, rotated rx 180 ry 0 rz -180 deg; joints [-126.042, -52.465, -82.97, 62.597, 65.614, -38.534]
  Call Extruder(403.79419)
  MoveL 8539 to (-39.1, 156.17, 125.68) mm, rotated rx 180 ry 0 rz 180 deg; joints [-126.05, -52.442, -83.021, 62.578, 65.623, -38.503]
  MoveL 8540 to (-39.1, 156.17, 125.68) mm, rotated rx 180 ry 0 rz 180 deg; joints [-126.05, -52.442, -83.021, 62.578, 65.623, -38.503]
  Call Extruder(403.97691)
  MoveL 8541 to (-39.22, 155.87, 125.68) mm, rotated rx 180 ry 0 rz 180 deg; joints [-126.06, -52.417, -83.081, 62.556, 65.632, -38.466]
  MoveL 8542 to (-39.22, 155.87, 125.68) mm, rotated rx 180 ry 0 rz 180 deg; joints [-126.06, -52.417, -83.081, 62.556, 65.632, -38.466]
  Call Extruder(404.15887)
  MoveL 8543 to (-39.35, 155.58, 125.68) mm, rotated rx -180 ry 0 rz 180 deg; joints [-126.07, -52.391, -83.14, 62.534, 65.642, -38.43]
  MoveL 8544 to (-39.35, 155.58, 125.68) mm, rotated rx -180 ry 0 rz 180 deg; joints [-126.07, -52.391, -83.14, 62.534, 65.642, -38.43]
  Call Extruder(404.30621)
  MoveL 8545 to (-39.44, 155.34, 125.68) mm, rotated rx 180 ry 0 rz 180 deg; joints [-126.079, -52.37, -83.188, 62.515, 65.649, -38.4]
  MoveL 8546 to (-39.44, 155.34, 125.68) mm, rotated rx 180 ry 0 rz 180 deg; joints [-126.079, -52.37, -83.188, 62.515, 65.649, -38.4]
  Call Extruder(404.41944)
  MoveL 8547 to (-39.5, 155.15, 125.68) mm, rotated rx 180 ry 0 rz 180 deg; joints [-126.087, -52.355, -83.225, 62.5, 65.653, -38.377]
  MoveL 8548 to (-39.5, 155.15, 125.68) mm, rotated rx 180 ry 0 rz 180 deg; joints [-126.087, -52.355, -83.225, 62.5, 65.653, -38.377]
  Call Extruder(404.53223)
  MoveL 8549 to (-39.56, 154.97, 125.68) mm, rotated rx -180 ry 0 rz 180 deg; joints [-126.095, -52.339, -83.261, 62.485, 65.658, -38.354]
  MoveL 8550 to (-39.56, 154.97, 125.68) mm, rotated rx -180 ry 0 rz 180 deg; joints [-126.095, -52.339, -83.261, 62.485, 65.658, -38.354]
  Call Extruder(404.64458)
  MoveL 8551 to (-39.62, 154.78, 125.68) mm, rotated rx 180 ry 0 rz 180 deg; joints [-126.103, -52.323, -83.297, 62.469, 65.662, -38.331]
  MoveL 8552 to (-39.62, 154.78, 125.68) mm, rotated rx 180 ry 0 rz 180 deg; joints [-126.103, -52.323, -83.297, 62.469, 65.662, -38.331]
  Call Extruder(404.75648)
  MoveL 8553 to (-39.68, 154.59, 125.68) mm, rotated rx 180 ry 0 rz 180 deg; joints [-126.111, -52.308, -83.334, 62.454, 65.667, -38.308]
  MoveL 8554 to (-39.68, 154.59, 125.68) mm, rotated rx 180 ry 0 rz 180 deg; joints [-126.111, -52.308, -83.334, 62.454, 65.667, -38.308]
  Call Extruder(404.87788)
  MoveL 8555 to (-39.75, 154.38, 125.68) mm, rotated rx 180 ry 0 rz 180 deg; joints [-126.12, -52.291, -83.373, 62.437, 65.671, -38.283]
  MoveL 8556 to (-39.75, 154.38, 125.68) mm, rotated rx 180 ry 0 rz 180 deg; joints [-126.12, -52.291, -83.373, 62.437, 65.671, -38.283]
  Call Extruder(405.00867)
  MoveL 8557 to (-39.82, 154.16, 125.68) mm, rotated rx 180 ry 0 rz 180 deg; joints [-126.131, -52.272, -83.416, 62.419, 65.676, -38.256]
  MoveL 8558 to (-39.82, 154.16, 125.68) mm, rotated rx 180 ry 0 rz 180 deg; joints [-126.131, -52.272, -83.416, 62.419, 65.676, -38.256]
  Call Extruder(405.13890)
  MoveL 8559 to (-39.88, 153.94, 125.68) mm, rotated rx -180 ry 0 rz -180 deg; joints [-126.141, -52.254, -83.458, 62.4, 65.681, -38.229]
  MoveL 8560 to (-39.88, 153.94, 125.68) mm, rotated rx -180 ry 0 rz -180 deg; joints [-126.141, -52.254, -83.458, 62.4, 65.681, -38.229]
  Call Extruder(405.26856)
  MoveL 8561 to (-39.95, 153.71, 125.68) mm, rotated rx 180 ry 0 rz -180 deg; joints [-126.151, -52.236, -83.501, 62.382, 65.686, -38.202]
  MoveL 8562 to (-39.95, 153.71, 125.68) mm, rotated rx 180 ry 0 rz -180 deg; joints [-126.151, -52.236, -83.501, 62.382, 65.686, -38.202]
  Call Extruder(405.39766)
  MoveL 8563 to (-40.02, 153.49, 125.68) mm, rotated rx -180 ry 0 rz -180 deg; joints [-126.161, -52.217, -83.543, 62.363, 65.691, -38.174]
  MoveL 8564 to (-40.02, 153.49, 125.68) mm, rotated rx -180 ry 0 rz -180 deg; joints [-126.161, -52.217, -83.543, 62.363, 65.691, -38.174]
  Call Extruder(405.51275)
  MoveL 8565 to (-40.06, 153.28, 125.68) mm, rotated rx -180 ry 0 rz 180 deg; joints [-126.173, -52.202, -83.58, 62.345, 65.694, -38.15]
  MoveL 8566 to (-40.06, 153.28, 125.68) mm, rotated rx -180 ry 0 rz 180 deg; joints [-126.173, -52.202, -83.58, 62.345, 65.694, -38.15]
  Call Extruder(405.62739)
  MoveL 8567 to (-40.11, 153.08, 125.68) mm, rotated rx 180 ry 0 rz 180 deg; joints [-126.184, -52.186, -83.617, 62.327, 65.697, -38.126]
  MoveL 8568 to (-40.11, 153.08, 125.68) mm, rotated rx 180 ry 0 rz 180 deg; joints [-126.184, -52.186, -83.617, 62.327, 65.697, -38.126]
  Call Extruder(405.74157)
  MoveL 8569 to (-40.15, 152.88, 125.68) mm, rotated rx 180 ry 0 rz 180 deg; joints [-126.195, -52.17, -83.654, 62.309, 65.699, -38.101]
  MoveL 8570 to (-40.15, 152.88, 125.68) mm, rotated rx 180 ry 0 rz 180 deg; joints [-126.195, -52.17, -83.654, 62.309, 65.699, -38.101]
  Call Extruder(405.85530)
  MoveL 8571 to (-40.2, 152.67, 125.68) mm, rotated rx -180 ry 0 rz 180 deg; joints [-126.206, -52.154, -83.691, 62.291, 65.702, -38.077]
  MoveL 8572 to (-40.2, 152.67, 125.68) mm, rotated rx -180 ry 0 rz 180 deg; joints [-126.206, -52.154, -83.691, 62.291, 65.702, -38.077]
  Call Extruder(405.98072)
  MoveL 8573 to (-40.24, 152.44, 125.68) mm, rotated rx 180 ry 0 rz 180 deg; joints [-126.219, -52.137, -83.731, 62.27, 65.705, -38.05]
  MoveL 8574 to (-40.24, 152.44, 125.68) mm, rotated rx 180 ry 0 rz 180 deg; joints [-126.219, -52.137, -83.731, 62.27, 65.705, -38.05]
  Call Extruder(406.11770)
  MoveL 8575 to (-40.29, 152.2, 125.68) mm, rotated rx 180 ry 0 rz 180 deg; joints [-126.233, -52.118, -83.776, 62.248, 65.708, -38.02]
  MoveL 8576 to (-40.29, 152.2, 125.68) mm, rotated rx 180 ry 0 rz 180 deg; joints [-126.233, -52.118, -83.776, 62.248, 65.708, -38.02]
  Call Extruder(406.25406)
  MoveL 8577 to (-40.34, 151.95, 125.68) mm, rotated rx -180 ry 0 rz 180 deg; joints [-126.248, -52.098, -83.82, 62.226, 65.711, -37.991]
  MoveL 8578 to (-40.34, 151.95, 125.68) mm, rotated rx -180 ry 0 rz 180 deg; joints [-126.248, -52.098, -83.82, 62.226, 65.711, -37.991]
  Call Extruder(406.38982)
  MoveL 8579 to (-40.39, 151.7, 125.68) mm, rotated rx 180 ry 0 rz 180 deg; joints [-126.262, -52.079, -83.864, 62.203, 65.714, -37.961]
  MoveL 8580 to (-40.39, 151.7, 125.68) mm, rotated rx 180 ry 0 rz 180 deg; joints [-126.262, -52.079, -83.864, 62.203, 65.714, -37.961]
  Call Extruder(406.52496)
  MoveL 8581 to (-40.44, 151.45, 125.68) mm, rotated rx 180 ry 0 rz -180 deg; joints [-126.276, -52.06, -83.908, 62.181, 65.717, -37.931]
  MoveL 8582 to (-40.44, 151.45, 125.68) mm, rotated rx 180 ry 0 rz -180 deg; joints [-126.276, -52.06, -83.908, 62.181, 65.717, -37.931]
  Call Extruder(406.65950)
  MoveL 8583 to (-40.49, 151.2, 125.68) mm, rotated rx 180 ry 0 rz 180 deg; joints [-126.291, -52.041, -83.953, 62.158, 65.72, -37.902]
  MoveL 8584 to (-40.49, 151.2, 125.68) mm, rotated rx 180 ry 0 rz 180 deg; joints [-126.291, -52.041, -83.953, 62.158, 65.72, -37.902]
  Call Extruder(406.79342)
  MoveL 8585 to (-40.54, 150.95, 125.68) mm, rotated rx 180 ry 0 rz 180 deg; joints [-126.305, -52.023, -83.997, 62.136, 65.723, -37.872]
  MoveL 8586 to (-40.54, 150.95, 125.68) mm, rotated rx 180 ry 0 rz 180 deg; joints [-126.305, -52.023, -83.997, 62.136, 65.723, -37.872]
  Call Extruder(406.94128)
  MoveL 8587 to (-40.59, 150.67, 125.68) mm, rotated rx 180 ry 0 rz 180 deg; joints [-126.322, -52.002, -84.045, 62.11, 65.725, -37.84]
  MoveL 8588 to (-40.59, 150.67, 125.68) mm, rotated rx 180 ry 0 rz 180 deg; joints [-126.322, -52.002, -84.045, 62.11, 65.725, -37.84]
  Call Extruder(407.10301)
  MoveL 8589 to (-40.64, 150.37, 125.68) mm, rotated rx -180 ry 0 rz 180 deg; joints [-126.341, -51.979, -84.098, 62.082, 65.728, -37.804]
  MoveL 8590 to (-40.64, 150.37, 125.68) mm, rotated rx -180 ry 0 rz 180 deg; joints [-126.341, -51.979, -84.098, 62.082, 65.728, -37.804]
  Call Extruder(407.26400)
  MoveL 8591 to (-40.69, 150.06, 125.68) mm, rotated rx -180 ry 0 rz 180 deg; joints [-126.36, -51.956, -84.151, 62.053, 65.73, -37.768]
  MoveL 8592 to (-40.69, 150.06, 125.68) mm, rotated rx -180 ry 0 rz 180 deg; joints [-126.36, -51.956, -84.151, 62.053, 65.73, -37.768]
  Call Extruder(407.42427)
  MoveL 8593 to (-40.74, 149.76, 125.68) mm, rotated rx -180 ry 0 rz 180 deg; joints [-126.379, -51.934, -84.203, 62.025, 65.733, -37.732]
  MoveL 8594 to (-40.74, 149.76, 125.68) mm, rotated rx -180 ry 0 rz 180 deg; joints [-126.379, -51.934, -84.203, 62.025, 65.733, -37.732]
  Call Extruder(407.58382)
  MoveL 8595 to (-40.78, 149.45, 125.68) mm, rotated rx -180 ry 0 rz 180 deg; joints [-126.398, -51.911, -84.256, 61.996, 65.735, -37.696]
  MoveL 8596 to (-40.78, 149.45, 125.68) mm, rotated rx -180 ry 0 rz 180 deg; joints [-126.398, -51.911, -84.256, 61.996, 65.735, -37.696]
  Call Extruder(407.74263)
  MoveL 8597 to (-40.83, 149.14, 125.68) mm, rotated rx -180 ry 0 rz 180 deg; joints [-126.417, -51.889, -84.309, 61.968, 65.738, -37.66]
  MoveL 8598 to (-40.83, 149.14, 125.68) mm, rotated rx -180 ry 0 rz 180 deg; joints [-126.417, -51.889, -84.309, 61.968, 65.738, -37.66]
  Call Extruder(407.92129)
  MoveL 8599 to (-40.88, 148.8, 125.68) mm, rotated rx 180 ry 0 rz 180 deg; joints [-126.439, -51.864, -84.367, 61.935, 65.74, -37.619]
  MoveL 8600 to (-40.88, 148.8, 125.68) mm, rotated rx 180 ry 0 rz 180 deg; joints [-126.439, -51.864, -84.367, 61.935, 65.74, -37.619]
  Call Extruder(408.11974)
  MoveL 8601 to (-40.92, 148.41, 125.68) mm, rotated rx 180 ry 0 rz 180 deg; joints [-126.465, -51.836, -84.432, 61.898, 65.741, -37.574]
  MoveL 8602 to (-40.92, 148.41, 125.68) mm, rotated rx 180 ry 0 rz 180 deg; joints [-126.465, -51.836, -84.432, 61.898, 65.741, -37.574]
  Call Extruder(408.31731)
  MoveL 8603 to (-40.97, 148.02, 125.68) mm, rotated rx -180 ry 0 rz 180 deg; joints [-126.491, -51.808, -84.497, 61.86, 65.743, -37.529]
  MoveL 8604 to (-40.97, 148.02, 125.68) mm, rotated rx -180 ry 0 rz 180 deg; joints [-126.491, -51.808, -84.497, 61.86, 65.743, -37.529]
  Call Extruder(408.51402)
  MoveL 8605 to (-41.02, 147.63, 125.68) mm, rotated rx -180 ry 0 rz 180 deg; joints [-126.517, -51.78, -84.562, 61.823, 65.745, -37.484]
  MoveL 8606 to (-41.02, 147.63, 125.68) mm, rotated rx -180 ry 0 rz 180 deg; joints [-126.517, -51.78, -84.562, 61.823, 65.745, -37.484]
  Call Extruder(408.70985)
  MoveL 8607 to (-41.06, 147.25, 125.68) mm, rotated rx -180 ry 0 rz 180 deg; joints [-126.543, -51.753, -84.627, 61.786, 65.746, -37.439]
  MoveL 8608 to (-41.06, 147.25, 125.68) mm, rotated rx -180 ry 0 rz 180 deg; joints [-126.543, -51.753, -84.627, 61.786, 65.746, -37.439]
  Call Extruder(409.00525)
  MoveL 8609 to (-41.11, 146.66, 125.68) mm, rotated rx 180 ry 0 rz -180 deg; joints [-126.585, -51.712, -84.722, 61.727, 65.747, -37.371]
  MoveL 8610 to (-41.11, 146.66, 125.68) mm, rotated rx 180 ry 0 rz -180 deg; joints [-126.585, -51.712, -84.722, 61.727, 65.747, -37.371]
  Call Extruder(409.29932)
  MoveL 8611 to (-41.16, 146.07, 125.68) mm, rotated rx -180 ry 0 rz -180 deg; joints [-126.628, -51.671, -84.818, 61.668, 65.747, -37.303]
  MoveL 8612 to (-41.16, 146.07, 125.68) mm, rotated rx -180 ry 0 rz -180 deg; joints [-126.628, -51.671, -84.818, 61.668, 65.747, -37.303]
  Call Extruder(409.59205)
  MoveL 8613 to (-41.2, 145.48, 125.68) mm, rotated rx -180 ry 0 rz 180 deg; joints [-126.67, -51.63, -84.913, 61.61, 65.747, -37.235]
  MoveL 8614 to (-41.2, 145.48, 125.68) mm, rotated rx -180 ry 0 rz 180 deg; joints [-126.67, -51.63, -84.913, 61.61, 65.747, -37.235]
  Call Extruder(410.16551)
  MoveL 8615 to (-41.25, 144.32, 125.68) mm, rotated rx 180 ry 0 rz 180 deg; joints [-126.759, -51.552, -85.096, 61.49, 65.743, -37.102]
  MoveL 8616 to (-41.25, 144.32, 125.68) mm, rotated rx 180 ry 0 rz 180 deg; joints [-126.759, -51.552, -85.096, 61.49, 65.743, -37.102]
  Call Extruder(410.87946)
  MoveL 8617 to (-41.29, 142.86, 125.68) mm, rotated rx 180 ry 0 rz -180 deg; joints [-126.873, -51.456, -85.322, 61.339, 65.737, -36.936]
  Call Extruder(452.94428)
  MoveL 8618 to (-41.29, 57.14, 125.68) mm, rotated rx -180 ry 0 rz 180 deg; joints [-135.148, -46.662, -97.084, 50.972, 65.214, -27.348]
  Call Extruder(453.37284)
  MoveL 8619 to (-41.27, 56.26, 125.68) mm, rotated rx 180 ry 0 rz -180 deg; joints [-135.25, -46.622, -97.189, 50.85, 65.208, -27.251]
  MoveL 8620 to (-41.27, 56.26, 125.68) mm, rotated rx 180 ry 0 rz -180 deg; joints [-135.25, -46.622, -97.189, 50.85, 65.208, -27.251]
  Call Extruder(453.94629)
  MoveL 8621 to (-41.22, 55.1, 125.68) mm, rotated rx 180 ry 0 rz 180 deg; joints [-135.387, -46.57, -97.325, 50.685, 65.198, -27.123]
  MoveL 8622 to (-41.22, 55.1, 125.68) mm, rotated rx 180 ry 0 rz 180 deg; joints [-135.387, -46.57, -97.325, 50.685, 65.198, -27.123]
  Call Extruder(454.38061)
  MoveL 8623 to (-41.18, 54.23, 125.68) mm, rotated rx -180 ry 0 rz 180 deg; joints [-135.493, -46.531, -97.426, 50.559, 65.189, -27.026]
  MoveL 8624 to (-41.18, 54.23, 125.68) mm, rotated rx -180 ry 0 rz 180 deg; joints [-135.493, -46.531, -97.426, 50.559, 65.189, -27.026]
  Call Extruder(454.67467)
  MoveL 8625 to (-41.13, 53.64, 125.68) mm, rotated rx 180 ry 0 rz 180 deg; joints [-135.566, -46.505, -97.492, 50.472, 65.182, -26.962]
  MoveL 8626 to (-41.13, 53.64, 125.68) mm, rotated rx 180 ry 0 rz 180 deg; joints [-135.566, -46.505, -97.492, 50.472, 65.182, -26.962]
  Call Extruder(454.97007)
  MoveL 8627 to (-41.09, 53.05, 125.68) mm, rotated rx 180 ry 0 rz 180 deg; joints [-135.64, -46.48, -97.558, 50.386, 65.174, -26.897]
  MoveL 8628 to (-41.09, 53.05, 125.68) mm, rotated rx 180 ry 0 rz 180 deg; joints [-135.64, -46.48, -97.558, 50.386, 65.174, -26.897]
  Call Extruder(455.21630)
  MoveL 8629 to (-41.04, 52.56, 125.68) mm, rotated rx 180 ry 0 rz 180 deg; joints [-135.701, -46.46, -97.611, 50.314, 65.167, -26.844]
  MoveL 8630 to (-41.04, 52.56, 125.68) mm, rotated rx 180 ry 0 rz 180 deg; joints [-135.701, -46.46, -97.611, 50.314, 65.167, -26.844]
  Call Extruder(455.41301)
  MoveL 8631 to (-40.99, 52.17, 125.68) mm, rotated rx 180 ry 0 rz 180 deg; joints [-135.751, -46.444, -97.652, 50.256, 65.161, -26.802]
  MoveL 8632 to (-40.99, 52.17, 125.68) mm, rotated rx 180 ry 0 rz 180 deg; joints [-135.751, -46.444, -97.652, 50.256, 65.161, -26.802]
  Call Extruder(455.61058)
  MoveL 8633 to (-40.95, 51.78, 125.68) mm, rotated rx -180 ry 0 rz 180 deg; joints [-135.801, -46.428, -97.693, 50.197, 65.155, -26.76]
  MoveL 8634 to (-40.95, 51.78, 125.68) mm, rotated rx -180 ry 0 rz 180 deg; joints [-135.801, -46.428, -97.693, 50.197, 65.155, -26.76]
  Call Extruder(455.80903)
  MoveL 8635 to (-40.9, 51.4, 125.68) mm, rotated rx 180 ry 0 rz -180 deg; joints [-135.852, -46.413, -97.734, 50.139, 65.148, -26.718]
  MoveL 8636 to (-40.9, 51.4, 125.68) mm, rotated rx 180 ry 0 rz -180 deg; joints [-135.852, -46.413, -97.734, 50.139, 65.148, -26.718]
  Call Extruder(456.00833)
  MoveL 8637 to (-40.86, 51.01, 125.68) mm, rotated rx 180 ry 0 rz 180 deg; joints [-135.902, -46.397, -97.775, 50.08, 65.142, -26.675]
  MoveL 8638 to (-40.86, 51.01, 125.68) mm, rotated rx 180 ry 0 rz 180 deg; joints [-135.902, -46.397, -97.775, 50.08, 65.142, -26.675]
  Call Extruder(456.16715)
  MoveL 8639 to (-40.81, 50.7, 125.68) mm, rotated rx 180 ry 0 rz -180 deg; joints [-135.943, -46.385, -97.806, 50.033, 65.136, -26.642]
  MoveL 8640 to (-40.81, 50.7, 125.68) mm, rotated rx 180 ry 0 rz -180 deg; joints [-135.943, -46.385, -97.806, 50.033, 65.136, -26.642]
  Call Extruder(456.32669)
  MoveL 8641 to (-40.76, 50.4, 125.68) mm, rotated rx 180 ry 0 rz -180 deg; joints [-135.984, -46.373, -97.836, 49.986, 65.129, -26.609]
  MoveL 8642 to (-40.76, 50.4, 125.68) mm, rotated rx 180 ry 0 rz -180 deg; joints [-135.984, -46.373, -97.836, 49.986, 65.129, -26.609]
  Call Extruder(456.48696)
  MoveL 8643 to (-40.71, 50.09, 125.68) mm, rotated rx 180 ry 0 rz -180 deg; joints [-136.025, -46.362, -97.867, 49.939, 65.123, -26.576]
  MoveL 8644 to (-40.71, 50.09, 125.68) mm, rotated rx 180 ry 0 rz -180 deg; joints [-136.025, -46.362, -97.867, 49.939, 65.123, -26.576]
  Call Extruder(456.64796)
  MoveL 8645 to (-40.66, 49.79, 125.68) mm, rotated rx -180 ry 0 rz -180 deg; joints [-136.067, -46.35, -97.898, 49.891, 65.117, -26.543]
  MoveL 8646 to (-40.66, 49.79, 125.68) mm, rotated rx -180 ry 0 rz -180 deg; joints [-136.067, -46.35, -97.898, 49.891, 65.117, -26.543]
  Call Extruder(456.80968)
